LIN {X 0,Y 227.887,Z 377.096,A -85,B 0,C 180,E1 -20034.128,E2 -20034.128} C_VEL
LIN {X 0,Y 227.876,Z 377.099,A -85,B 0,C 180,E1 -20038.377,E2 -20038.377} C_VEL
LIN {X 0,Y 227.892,Z 377.098,A -85,B 0,C 180,E1 -20042.444,E2 -20042.444} C_VEL
LIN {X 0,Y 227.92,Z 377.094,A -85,B 0,C 180,E1 -20046.367,E2 -20046.367} C_VEL
LIN {X 0,Y 228.003,Z 377.201,A -85,B 0,C 180,E1 -20049.532,E2 -20049.532} C_VEL
LIN {X 0,Y 229.065,Z 380.026,A -85,B 0,C 180,E1 -20049.897,E2 -20049.897} C_VEL
LIN {X 0,Y 233.26,Z 390.63,A -85,B 0,C 180,E1 -20051.459,E2 -20051.459} C_VEL
LIN {X 0,Y 236.547,Z 400.917,A -85,B 0,C 180,E1 -20053.149,E2 -20053.149} C_VEL
LIN {X 0,Y 238.293,Z 407.679,A -85,B 0,C 180,E1 -20054.381,E2 -20054.381} C_VEL
LIN {X 0,Y 236.571,Z 418.908,A -85,B 0,C 180,E1 -20056.25,E2 -20056.25} C_VEL
LIN {X 0,Y 234.854,Z 428.795,A -85,B 0,C 180,E1 -20058.345,E2 -20058.345} C_VEL
LIN {X 0,Y 232.986,Z 438.362,A -85,B 0,C 180,E1 -20060.887,E2 -20060.887} C_VEL
LIN {X 0,Y 231.325,Z 446.044,A -85,B 0,C 180,E1 -20063.457,E2 -20063.457} C_VEL
LIN {X 0,Y 230.205,Z 451.273,A -85,B 0,C 180,E1 -20065.621,E2 -20065.621} C_VEL
LIN {X 0,Y 229.202,Z 456.365,A -85,B 0,C 180,E1 -20068.242,E2 -20068.242} C_VEL
LIN {X 0,Y 228.364,Z 460.351,A -85,B 0,C 180,E1 -20070.88,E2 -20070.88} C_VEL
LIN {X 0,Y 227.825,Z 463.315,A -85,B 0,C 180,E1 -20073.536,E2 -20073.536} C_VEL
LIN {X 0,Y 227.82,Z 464.727,A -85,B 0,C 180,E1 -20075.309,E2 -20075.309} C_VEL
LIN {X 0,Y 227.806,Z 465.754,A -85,B 0,C 180,E1 -20077.087,E2 -20077.087} C_VEL
LIN {X 0,Y 227.876,Z 466.526,A -85,B 0,C 180,E1 -20079.272,E2 -20079.272} C_VEL
LIN {X 0,Y 228.342,Z 466.545,A -85,B 0,C 180,E1 -20082.441,E2 -20082.441} C_VEL
LIN {X 0,Y 229.386,Z 465.08,A -85,B 0,C 180,E1 -20086.005,E2 -20086.005} C_VEL
LIN {X 0,Y 230.21,Z 463.745,A -85,B 0,C 180,E1 -20087.774,E2 -20087.774} C_VEL
LIN {X 0,Y 231.644,Z 460.912,A -85,B 0,C 180,E1 -20090.419,E2 -20090.419} C_VEL
LIN {X 0,Y 233.383,Z 457.03,A -85,B 0,C 180,E1 -20093.045,E2 -20093.045} C_VEL
LIN {X 0,Y 235.482,Z 451.966,A -85,B 0,C 180,E1 -20095.641,E2 -20095.641} C_VEL
LIN {X 0,Y 237.977,Z 445.525,A -85,B 0,C 180,E1 -20098.196,E2 -20098.196} C_VEL
LIN {X 0,Y 240.822,Z 437.456,A -85,B 0,C 180,E1 -20100.71,E2 -20100.71} C_VEL
LIN {X 0,Y 243.404,Z 429.151,A -85,B 0,C 180,E1 -20102.776,E2 -20102.776} C_VEL
LIN {X 0,Y 245.548,Z 421.099,A -85,B 0,C 180,E1 -20104.42,E2 -20104.42} C_VEL
LIN {X 0,Y 243.299,Z 411.924,A -85,B 0,C 180,E1 -20106.717,E2 -20106.717} C_VEL
LIN {X 0,Y 240.025,Z 402.244,A -85,B 0,C 180,E1 -20108.979,E2 -20108.979} C_VEL
LIN {X 0,Y 235.855,Z 392.708,A -85,B 0,C 180,E1 -20111.136,E2 -20111.136} C_VEL
LIN {X 0,Y 231.014,Z 383.649,A -85,B 0,C 180,E1 -20113.173,E2 -20113.173} C_VEL
LIN {X 0,Y 229.588,Z 380.946,A -85,B 0,C 180,E1 -20113.738,E2 -20113.738} C_VEL
LIN {X 0,Y 228.183,Z 378.565,A -85,B 0,C 180,E1 -20114.266,E2 -20114.266} C_VEL
LIN {X 0,Y 227.841,Z 377.102,A -85,B 0,C 180,E1 -20114.494,E2 -20114.494} C_VEL
LIN {X 0,Y 227.866,Z 377.101,A -85,B 0,C 180,E1 -20117.748,E2 -20117.748} C_VEL
LIN {X 0,Y 227.87,Z 377.105,A -85,B 0,C 180,E1 -20121.913,E2 -20121.913} C_VEL
LIN {X 0,Y 227.889,Z 377.096,A -85,B 0,C 180,E1 -20126.371,E2 -20126.371} C_VEL
LIN {X 0,Y 227.902,Z 377.05,A -85,B 0,C 180,E1 -20130.435,E2 -20130.435} C_VEL
LIN {X 0,Y 227.926,Z 377.093,A -85,B 0,C 180,E1 -20134.425,E2 -20134.425} C_VEL
LIN {X 0,Y 227.959,Z 377.082,A -85,B 0,C 180,E1 -20138.286,E2 -20138.286} C_VEL
LIN {X 0,Y 228.031,Z 377.067,A -85,B 0,C 180,E1 -20142.825,E2 -20142.825} C_VEL
LIN {X 0,Y 228.091,Z 377.072,A -85,B 0,C 180,E1 -20147.544,E2 -20147.544} C_VEL
LIN {X 0,Y 228.322,Z 377.045,A -85,B 0,C 180,E1 -20151.146,E2 -20151.146} C_VEL
LIN {X 0,Y 228.355,Z 377.031,A -85,B 0,C 180,E1 -20152.928,E2 -20152.928} C_VEL
LIN {X 0,Y 228.554,Z 377.012,A -85,B 0,C 180,E1 -20158.237,E2 -20158.237} C_VEL
LIN {X 0,Y 228.554,Z 377.013,A -85,B 0,C 180,E1 -20161.762,E2 -20161.762} C_VEL
LIN {X 0,Y 228.355,Z 377.04,A -85,B 0,C 180,E1 -20167.071,E2 -20167.071} C_VEL
LIN {X 0,Y 228.167,Z 377.054,A -85,B 0,C 180,E1 -20170.65,E2 -20170.65} C_VEL
LIN {X 0,Y 228.053,Z 377.078,A -85,B 0,C 180,E1 -20176.102,E2 -20176.102} C_VEL
LIN {X 0,Y 227.939,Z 377.091,A -85,B 0,C 180,E1 -20179.825,E2 -20179.825} C_VEL
LIN {X 0,Y 227.91,Z 377.093,A -85,B 0,C 180,E1 -20183.633,E2 -20183.633} C_VEL
LIN {X 0,Y 227.9,Z 377.101,A -85,B 0,C 180,E1 -20188.177,E2 -20188.177} C_VEL
LIN {X 0,Y 228.571,Z 380.288,A -85,B 0,C 180,E1 -20191.514,E2 -20191.514} C_VEL
LIN {X 0,Y 229.542,Z 384.592,A -85,B 0,C 180,E1 -20195.572,E2 -20195.572} C_VEL
LIN {X 0,Y 230.655,Z 390.276,A -85,B 0,C 180,E1 -20200.384,E2 -20200.384} C_VEL
LIN {X 0,Y 231.787,Z 396.318,A -85,B 0,C 180,E1 -20205.043,E2 -20205.043} C_VEL
LIN {X 0,Y 232.75,Z 401.888,A -85,B 0,C 180,E1 -20209.015,E2 -20209.015} C_VEL
LIN {X 0,Y 232.897,Z 404.605,A -85,B 0,C 180,E1 -20210.825,E2 -20210.825} C_VEL
LIN {X 0,Y 231.681,Z 409.325,A -85,B 0,C 180,E1 -20213.706,E2 -20213.706} C_VEL
LIN {X 0,Y 232.555,Z 412.987,A -85,B 0,C 180,E1 -20214.055,E2 -20214.055} C_VEL
LIN {X 0,Y 233.833,Z 417.977,A -85,B 0,C 180,E1 -20214.599,E2 -20214.599} C_VEL
LIN {X 0,Y 234.21,Z 423.584,A -85,B 0,C 180,E1 -20215.071,E2 -20215.071} C_VEL
LIN {X 0,Y 233.3,Z 433.06,A -85,B 0,C 180,E1 -20215.782,E2 -20215.782} C_VEL
LIN {X 0,Y 232.111,Z 442.304,A -85,B 0,C 180,E1 -20216.645,E2 -20216.645} C_VEL
LIN {X 0,Y 232.068,Z 447.482,A -85,B 0,C 180,E1 -20217.347,E2 -20217.347} C_VEL
LIN {X 0,Y 232.339,Z 459.542,A -85,B 0,C 180,E1 -20219.308,E2 -20219.308} C_VEL
LIN {X 0,Y 231.84,Z 470.153,A -85,B 0,C 180,E1 -20221.291,E2 -20221.291} C_VEL
LIN {X 0,Y 230.723,Z 479.469,A -85,B 0,C 180,E1 -20223.303,E2 -20223.303} C_VEL
LIN {X 0,Y 228.773,Z 488.259,A -85,B 0,C 180,E1 -20225.499,E2 -20225.499} C_VEL
LIN {X 0,Y 225.7,Z 496.785,A -85,B 0,C 180,E1 -20228.06,E2 -20228.06} C_VEL
LIN {X 0,Y 223.14,Z 504.144,A -85,B 0,C 180,E1 -20230.887,E2 -20230.887} C_VEL
LIN {X 0,Y 221.5,Z 509.326,A -85,B 0,C 180,E1 -20233.409,E2 -20233.409} C_VEL
LIN {X 0,Y 220.196,Z 513.777,A -85,B 0,C 180,E1 -20236.152,E2 -20236.152} C_VEL
LIN {X 0,Y 219.485,Z 517.195,A -85,B 0,C 180,E1 -20238.925,E2 -20238.925} C_VEL
LIN {X 0,Y 219.334,Z 520.299,A -85,B 0,C 180,E1 -20242.637,E2 -20242.637} C_VEL
LIN {X 0,Y 219.825,Z 521.726,A -85,B 0,C 180,E1 -20246.335,E2 -20246.335} C_VEL
LIN {X 0,Y 220.089,Z 521.828,A -85,B 0,C 180,E1 -20248.171,E2 -20248.171} C_VEL
LIN {X 0,Y 220.231,Z 521.508,A -85,B 0,C 180,E1 -20250.001,E2 -20250.001} C_VEL
LIN {X 0,Y 220.159,Z 520.712,A -85,B 0,C 180,E1 -20251.831,E2 -20251.831} C_VEL
LIN {X 0,Y 219.982,Z 519.453,A -85,B 0,C 180,E1 -20253.665,E2 -20253.665} C_VEL
LIN {X 0,Y 219.583,Z 515.837,A -85,B 0,C 180,E1 -20257.166,E2 -20257.166} C_VEL
LIN {X 0,Y 219.532,Z 511.426,A -85,B 0,C 180,E1 -20260.143,E2 -20260.143} C_VEL
LIN {X 0,Y 220.146,Z 505.04,A -85,B 0,C 180,E1 -20263.384,E2 -20263.384} C_VEL
LIN {X 0,Y 221.1,Z 498.086,A -85,B 0,C 180,E1 -20266.15,E2 -20266.15} C_VEL
LIN {X 0,Y 222.436,Z 491.045,A -85,B 0,C 180,E1 -20268.42,E2 -20268.42} C_VEL
LIN {X 0,Y 224.159,Z 482.585,A -85,B 0,C 180,E1 -20270.655,E2 -20270.655} C_VEL
LIN {X 0,Y 224.752,Z 475.375,A -85,B 0,C 180,E1 -20272.282,E2 -20272.282} C_VEL
LIN {X 0,Y 225.233,Z 464.959,A -85,B 0,C 180,E1 -20274.281,E2 -20274.281} C_VEL
LIN {X 0,Y 225.518,Z 453.251,A -85,B 0,C 180,E1 -20276.117,E2 -20276.117} C_VEL
LIN {X 0,Y 225.191,Z 441.055,A -85,B 0,C 180,E1 -20277.662,E2 -20277.662} C_VEL
LIN {X 0,Y 224.037,Z 427.624,A -85,B 0,C 180,E1 -20279.036,E2 -20279.036} C_VEL
LIN {X 0,Y 221.953,Z 413.948,A -85,B 0,C 180,E1 -20280.141,E2 -20280.141} C_VEL
LIN {X 0,Y 221.507,Z 411.003,A -85,B 0,C 180,E1 -20280.389,E2 -20280.389} C_VEL
LIN {X 0,Y 223.273,Z 402.178,A -85,B 0,C 180,E1 -20285.733,E2 -20285.733} C_VEL
LIN {X 0,Y 224.225,Z 397.146,A -85,B 0,C 180,E1 -20288.821,E2 -20288.821} C_VEL
LIN {X 0,Y 223.836,Z 393.482,A -85,B 0,C 180,E1 -20291.253,E2 -20291.253} C_VEL
LIN {X 0,Y 222.551,Z 386.745,A -85,B 0,C 180,E1 -20295.993,E2 -20295.993} C_VEL
LIN {X 0,Y 221.357,Z 380.661,A -85,B 0,C 180,E1 -20300.581,E2 -20300.581} C_VEL
LIN {X 0,Y 220.858,Z 377.978,A -85,B 0,C 180,E1 -20302.8,E2 -20302.8} C_VEL
LIN {X 0,Y 220.821,Z 377.981,A -85,B 0,C 180,E1 -20307.245,E2 -20307.245} C_VEL
LIN {X 0,Y 220.832,Z 377.977,A -85,B 0,C 180,E1 -20311.486,E2 -20311.486} C_VEL
LIN {X 0,Y 220.873,Z 377.974,A -85,B 0,C 180,E1 -20315.566,E2 -20315.566} C_VEL
LIN {X 0,Y 220.898,Z 377.971,A -85,B 0,C 180,E1 -20319.515,E2 -20319.515} C_VEL
LIN {X 0,Y 221.022,Z 377.955,A -85,B 0,C 180,E1 -20323.371,E2 -20323.371} C_VEL
LIN {X 0,Y 221.123,Z 377.941,A -85,B 0,C 180,E1 -20329.007,E2 -20329.007} C_VEL
LIN {X 0,Y 221.317,Z 377.917,A -85,B 0,C 180,E1 -20332.703,E2 -20332.703} C_VEL
LIN {X 0,Y 221.518,Z 377.881,A -85,B 0,C 180,E1 -20338.182,E2 -20338.182} C_VEL
LIN {X 0,Y 221.519,Z 377.89,A -85,B 0,C 180,E1 -20341.819,E2 -20341.819} C_VEL
LIN {X 0,Y 221.302,Z 377.906,A -85,B 0,C 180,E1 -20347.298,E2 -20347.298} C_VEL
LIN {X 0,Y 221.123,Z 377.939,A -85,B 0,C 180,E1 -20350.994,E2 -20350.994} C_VEL
LIN {X 0,Y 221.023,Z 377.948,A -85,B 0,C 180,E1 -20356.63,E2 -20356.63} C_VEL
LIN {X 0,Y 220.9,Z 377.965,A -85,B 0,C 180,E1 -20360.486,E2 -20360.486} C_VEL
LIN {X 0,Y 220.874,Z 377.968,A -85,B 0,C 180,E1 -20364.435,E2 -20364.435} C_VEL
LIN {X 0,Y 220.842,Z 377.972,A -85,B 0,C 180,E1 -20368.513,E2 -20368.513} C_VEL
LIN {X 0,Y 220.831,Z 377.975,A -85,B 0,C 180,E1 -20372.754,E2 -20372.754} C_VEL
LIN {X 0,Y 220.844,Z 377.976,A -85,B 0,C 180,E1 -20377.288,E2 -20377.288} C_VEL
LIN {X 0,Y 220.782,Z 377.981,A -85,B 0,C 180,E1 -20381.951,E2 -20381.951} C_VEL
LIN {X 0,Y 220.781,Z 377.983,A -85,B 0,C 180,E1 -20385.546,E2 -20385.546} C_VEL
LIN {X 0,Y 220.812,Z 377.976,A -85,B 0,C 180,E1 -20390.463,E2 -20390.463} C_VEL
LIN {X 0,Y 220.807,Z 377.979,A -85,B 0,C 180,E1 -20395.045,E2 -20395.045} C_VEL
LIN {X 0,Y 220.874,Z 377.973,A -85,B 0,C 180,E1 -20399.394,E2 -20399.394} C_VEL
LIN {X 0,Y 220.901,Z 377.969,A -85,B 0,C 180,E1 -20403.549,E2 -20403.549} C_VEL
LIN {X 0,Y 220.95,Z 378.071,A -85,B 0,C 180,E1 -20408.665,E2 -20408.665} C_VEL
LIN {X 0,Y 222.527,Z 382.229,A -85,B 0,C 180,E1 -20409.233,E2 -20409.233} C_VEL
LIN {X 0,Y 226.794,Z 393.014,A -85,B 0,C 180,E1 -20410.941,E2 -20410.941} C_VEL
LIN {X 0,Y 229.89,Z 402.635,A -85,B 0,C 180,E1 -20412.622,E2 -20412.622} C_VEL
LIN {X 0,Y 231.599,Z 409.377,A -85,B 0,C 180,E1 -20413.906,E2 -20413.906} C_VEL
LIN {X 0,Y 229.783,Z 420.479,A -85,B 0,C 180,E1 -20415.836,E2 -20415.836} C_VEL
LIN {X 0,Y 227.986,Z 430.233,A -85,B 0,C 180,E1 -20417.989,E2 -20417.989} C_VEL
LIN {X 0,Y 226.054,Z 439.706,A -85,B 0,C 180,E1 -20420.605,E2 -20420.605} C_VEL
LIN {X 0,Y 224.343,Z 447.271,A -85,B 0,C 180,E1 -20423.252,E2 -20423.252} C_VEL
LIN {X 0,Y 223.197,Z 452.453,A -85,B 0,C 180,E1 -20425.484,E2 -20425.484} C_VEL
LIN {X 0,Y 222.17,Z 457.472,A -85,B 0,C 180,E1 -20428.186,E2 -20428.186} C_VEL
LIN {X 0,Y 221.304,Z 461.404,A -85,B 0,C 180,E1 -20430.908,E2 -20430.908} C_VEL
LIN {X 0,Y 220.773,Z 464.322,A -85,B 0,C 180,E1 -20433.649,E2 -20433.649} C_VEL
LIN {X 0,Y 220.786,Z 465.69,A -85,B 0,C 180,E1 -20435.478,E2 -20435.478} C_VEL
LIN {X 0,Y 220.813,Z 467.331,A -85,B 0,C 180,E1 -20439.156,E2 -20439.156} C_VEL
LIN {X 0,Y 221.027,Z 467.571,A -85,B 0,C 180,E1 -20440.997,E2 -20440.997} C_VEL
LIN {X 0,Y 221.9,Z 466.818,A -85,B 0,C 180,E1 -20444.676,E2 -20444.676} C_VEL
LIN {X 0,Y 222.53,Z 465.869,A -85,B 0,C 180,E1 -20446.512,E2 -20446.512} C_VEL
LIN {X 0,Y 224.288,Z 462.893,A -85,B 0,C 180,E1 -20449.94,E2 -20449.94} C_VEL
LIN {X 0,Y 226.142,Z 459.077,A -85,B 0,C 180,E1 -20452.858,E2 -20452.858} C_VEL
LIN {X 0,Y 228.246,Z 454.359,A -85,B 0,C 180,E1 -20455.535,E2 -20455.535} C_VEL
LIN {X 0,Y 230.688,Z 448.476,A -85,B 0,C 180,E1 -20458.118,E2 -20458.118} C_VEL
LIN {X 0,Y 233.681,Z 440.8,A -85,B 0,C 180,E1 -20460.748,E2 -20460.748} C_VEL
LIN {X 0,Y 236.769,Z 431.449,A -85,B 0,C 180,E1 -20463.243,E2 -20463.243} C_VEL
LIN {X 0,Y 239.085,Z 423.424,A -85,B 0,C 180,E1 -20464.972,E2 -20464.972} C_VEL
LIN {X 0,Y 237.322,Z 415.381,A -85,B 0,C 180,E1 -20467.097,E2 -20467.097} C_VEL
LIN {X 0,Y 234.296,Z 405.948,A -85,B 0,C 180,E1 -20469.464,E2 -20469.464} C_VEL
LIN {X 0,Y 230.508,Z 396.85,A -85,B 0,C 180,E1 -20471.669,E2 -20471.669} C_VEL
LIN {X 0,Y 225.272,Z 386.406,A -85,B 0,C 180,E1 -20474.146,E2 -20474.146} C_VEL
LIN {X 0,Y 223.216,Z 382.634,A -85,B 0,C 180,E1 -20475.019,E2 -20475.019} C_VEL
LIN {X 0,Y 221.246,Z 379.798,A -85,B 0,C 180,E1 -20475.769,E2 -20475.769} C_VEL
LIN {X 0,Y 220.79,Z 377.984,A -85,B 0,C 180,E1 -20476.07,E2 -20476.07} C_VEL
LIN {X 0,Y 220.848,Z 377.972,A -85,B 0,C 180,E1 -20480.471,E2 -20480.471} C_VEL
LIN {X 0,Y 220.814,Z 377.979,A -85,B 0,C 180,E1 -20485.047,E2 -20485.047} C_VEL
LIN {X 0,Y 220.831,Z 377.93,A -85,B 0,C 180,E1 -20489.389,E2 -20489.389} C_VEL
LIN {X 0,Y 220.892,Z 377.965,A -85,B 0,C 180,E1 -20493.548,E2 -20493.548} C_VEL
LIN {X 0,Y 220.875,Z 377.958,A -85,B 0,C 180,E1 -20497.553,E2 -20497.553} C_VEL
LIN {X 0,Y 220.981,Z 377.944,A -85,B 0,C 180,E1 -20502.57,E2 -20502.57} C_VEL
LIN {X 0,Y 221.023,Z 377.95,A -85,B 0,C 180,E1 -20507.139,E2 -20507.139} C_VEL
LIN {X 0,Y 221.255,Z 377.925,A -85,B 0,C 180,E1 -20510.861,E2 -20510.861} C_VEL
LIN {X 0,Y 221.308,Z 377.911,A -85,B 0,C 180,E1 -20512.702,E2 -20512.702} C_VEL
LIN {X 0,Y 221.512,Z 377.889,A -85,B 0,C 180,E1 -20518.181,E2 -20518.181} C_VEL
LIN {X 0,Y 221.512,Z 377.89,A -85,B 0,C 180,E1 -20521.818,E2 -20521.818} C_VEL
LIN {X 0,Y 221.307,Z 377.919,A -85,B 0,C 180,E1 -20527.297,E2 -20527.297} C_VEL
LIN {X 0,Y 221.113,Z 377.935,A -85,B 0,C 180,E1 -20530.994,E2 -20530.994} C_VEL
LIN {X 0,Y 221.012,Z 377.951,A -85,B 0,C 180,E1 -20536.63,E2 -20536.63} C_VEL
LIN {X 0,Y 220.889,Z 377.965,A -85,B 0,C 180,E1 -20540.486,E2 -20540.486} C_VEL
LIN {X 0,Y 220.863,Z 377.973,A -85,B 0,C 180,E1 -20544.435,E2 -20544.435} C_VEL
LIN {X 0,Y 220.882,Z 378.056,A -85,B 0,C 180,E1 -20547.016,E2 -20547.016} C_VEL
LIN {X 0,Y 221.685,Z 381.884,A -85,B 0,C 180,E1 -20551.136,E2 -20551.136} C_VEL
LIN {X 0,Y 222.721,Z 386.64,A -85,B 0,C 180,E1 -20555.715,E2 -20555.715} C_VEL
LIN {X 0,Y 223.697,Z 391.587,A -85,B 0,C 180,E1 -20560.046,E2 -20560.046} C_VEL
LIN {X 0,Y 224.796,Z 397.571,A -85,B 0,C 180,E1 -20564.817,E2 -20564.817} C_VEL
LIN {X 0,Y 225.818,Z 403.494,A -85,B 0,C 180,E1 -20569.191,E2 -20569.191} C_VEL
LIN {X 0,Y 225.941,Z 405.065,A -85,B 0,C 180,E1 -20570.283,E2 -20570.283} C_VEL
LIN {X 0,Y 225.199,Z 408.146,A -85,B 0,C 180,E1 -20572.279,E2 -20572.279} C_VEL
LIN {X 0,Y 226.113,Z 412.034,A -85,B 0,C 180,E1 -20572.703,E2 -20572.703} C_VEL
LIN {X 0,Y 229.199,Z 425.135,A -85,B 0,C 180,E1 -20574.279,E2 -20574.279} C_VEL
LIN {X 0,Y 231.364,Z 438.931,A -85,B 0,C 180,E1 -20576.106,E2 -20576.106} C_VEL
LIN {X 0,Y 232.068,Z 447.482,A -85,B 0,C 180,E1 -20577.347,E2 -20577.347} C_VEL
LIN {X 0,Y 232.005,Z 451.013,A -85,B 0,C 180,E1 -20577.851,E2 -20577.851} C_VEL
LIN {X 0,Y 230.913,Z 456.25,A -85,B 0,C 180,E1 -20578.526,E2 -20578.526} C_VEL
LIN {X 0,Y 229.109,Z 461.374,A -85,B 0,C 180,E1 -20579.176,E2 -20579.176} C_VEL
LIN {X 0,Y 226.008,Z 469.424,A -85,B 0,C 180,E1 -20580.386,E2 -20580.386} C_VEL
LIN {X 0,Y 224.98,Z 473.951,A -85,B 0,C 180,E1 -20581.289,E2 -20581.289} C_VEL
LIN {X 0,Y 223.536,Z 482.712,A -85,B 0,C 180,E1 -20583.385,E2 -20583.385} C_VEL
LIN {X 0,Y 221.75,Z 489.26,A -85,B 0,C 180,E1 -20585.171,E2 -20585.171} C_VEL
LIN {X 0,Y 218.628,Z 497.453,A -85,B 0,C 180,E1 -20587.809,E2 -20587.809} C_VEL
LIN {X 0,Y 216.24,Z 503.98,A -85,B 0,C 180,E1 -20590.48,E2 -20590.48} C_VEL
LIN {X 0,Y 214.129,Z 510.227,A -85,B 0,C 180,E1 -20593.802,E2 -20593.802} C_VEL
LIN {X 0,Y 212.898,Z 514.277,A -85,B 0,C 180,E1 -20596.641,E2 -20596.641} C_VEL
LIN {X 0,Y 212.25,Z 518.145,A -85,B 0,C 180,E1 -20600.472,E2 -20600.472} C_VEL
LIN {X 0,Y 212.351,Z 519.863,A -85,B 0,C 180,E1 -20603.159,E2 -20603.159} C_VEL
LIN {X 0,Y 212.748,Z 520.857,A -85,B 0,C 180,E1 -20606.213,E2 -20606.213} C_VEL
LIN {X 0,Y 213.035,Z 520.945,A -85,B 0,C 180,E1 -20608.111,E2 -20608.111} C_VEL
LIN {X 0,Y 213.184,Z 520.605,A -85,B 0,C 180,E1 -20610.001,E2 -20610.001} C_VEL
LIN {X 0,Y 213.108,Z 519.773,A -85,B 0,C 180,E1 -20611.891,E2 -20611.891} C_VEL
LIN {X 0,Y 212.904,Z 518.49,A -85,B 0,C 180,E1 -20613.787,E2 -20613.787} C_VEL
LIN {X 0,Y 212.506,Z 515.093,A -85,B 0,C 180,E1 -20617.179,E2 -20617.179} C_VEL
LIN {X 0,Y 212.5,Z 510.36,A -85,B 0,C 180,E1 -20620.482,E2 -20620.482} C_VEL
LIN {X 0,Y 213.188,Z 503.916,A -85,B 0,C 180,E1 -20623.829,E2 -20623.829} C_VEL
LIN {X 0,Y 214.218,Z 496.905,A -85,B 0,C 180,E1 -20626.684,E2 -20626.684} C_VEL
LIN {X 0,Y 215.928,Z 488.924,A -85,B 0,C 180,E1 -20629.285,E2 -20629.285} C_VEL
LIN {X 0,Y 217.407,Z 481.258,A -85,B 0,C 180,E1 -20631.327,E2 -20631.327} C_VEL
LIN {X 0,Y 218.032,Z 471.647,A -85,B 0,C 180,E1 -20633.51,E2 -20633.51} C_VEL
LIN {X 0,Y 218.596,Z 460.828,A -85,B 0,C 180,E1 -20635.521,E2 -20635.521} C_VEL
LIN {X 0,Y 218.745,Z 449.749,A -85,B 0,C 180,E1 -20637.221,E2 -20637.221} C_VEL
LIN {X 0,Y 218.234,Z 437.493,A -85,B 0,C 180,E1 -20638.775,E2 -20638.775} C_VEL
LIN {X 0,Y 217.001,Z 424.909,A -85,B 0,C 180,E1 -20640.073,E2 -20640.073} C_VEL
LIN {X 0,Y 214.936,Z 412.402,A -85,B 0,C 180,E1 -20641.11,E2 -20641.11} C_VEL
LIN {X 0,Y 214.672,Z 410.082,A -85,B 0,C 180,E1 -20641.307,E2 -20641.307} C_VEL
LIN {X 0,Y 216.59,Z 401.221,A -85,B 0,C 180,E1 -20646.893,E2 -20646.893} C_VEL
LIN {X 0,Y 217.178,Z 397.839,A -85,B 0,C 180,E1 -20649.045,E2 -20649.045} C_VEL
LIN {X 0,Y 216.714,Z 393.929,A -85,B 0,C 180,E1 -20651.765,E2 -20651.765} C_VEL
LIN {X 0,Y 215.394,Z 387.122,A -85,B 0,C 180,E1 -20656.749,E2 -20656.749} C_VEL
LIN {X 0,Y 214.269,Z 381.185,A -85,B 0,C 180,E1 -20661.45,E2 -20661.45} C_VEL
LIN {X 0,Y 213.765,Z 378.863,A -85,B 0,C 180,E1 -20663.49,E2 -20663.49} C_VEL
LIN {X 0,Y 213.772,Z 378.857,A -85,B 0,C 180,E1 -20668.263,E2 -20668.263} C_VEL
LIN {X 0,Y 213.831,Z 378.852,A -85,B 0,C 180,E1 -20672.604,E2 -20672.604} C_VEL
LIN {X 0,Y 213.857,Z 378.851,A -85,B 0,C 180,E1 -20676.954,E2 -20676.954} C_VEL
LIN {X 0,Y 213.938,Z 378.84,A -85,B 0,C 180,E1 -20682.306,E2 -20682.306} C_VEL
LIN {X 0,Y 213.987,Z 378.831,A -85,B 0,C 180,E1 -20686.709,E2 -20686.709} C_VEL
LIN {X 0,Y 214.203,Z 378.805,A -85,B 0,C 180,E1 -20690.558,E2 -20690.558} C_VEL
LIN {X 0,Y 214.254,Z 378.797,A -85,B 0,C 180,E1 -20692.461,E2 -20692.461} C_VEL
LIN {X 0,Y 214.452,Z 378.761,A -85,B 0,C 180,E1 -20698.122,E2 -20698.122} C_VEL
LIN {X 0,Y 214.557,Z 378.751,A -85,B 0,C 180,E1 -20700,E2 -20700} C_VEL
LIN {X 0,Y 214.452,Z 378.77,A -85,B 0,C 180,E1 -20701.878,E2 -20701.878} C_VEL
LIN {X 0,Y 214.242,Z 378.785,A -85,B 0,C 180,E1 -20707.54,E2 -20707.54} C_VEL
LIN {X 0,Y 214.054,Z 378.82,A -85,B 0,C 180,E1 -20711.362,E2 -20711.362} C_VEL
LIN {X 0,Y 213.94,Z 378.823,A -85,B 0,C 180,E1 -20715.237,E2 -20715.237} C_VEL
LIN {X 0,Y 213.847,Z 378.846,A -85,B 0,C 180,E1 -20719.187,E2 -20719.187} C_VEL
LIN {X 0,Y 213.854,Z 378.835,A -85,B 0,C 180,E1 -20723.227,E2 -20723.227} C_VEL
LIN {X 0,Y 213.835,Z 378.85,A -85,B 0,C 180,E1 -20727.45,E2 -20727.45} C_VEL
LIN {X 0,Y 213.786,Z 378.851,A -85,B 0,C 180,E1 -20731.735,E2 -20731.735} C_VEL
LIN {X 0,Y 213.759,Z 378.857,A -85,B 0,C 180,E1 -20736.286,E2 -20736.286} C_VEL
LIN {X 0,Y 213.724,Z 378.862,A -85,B 0,C 180,E1 -20741.123,E2 -20741.123} C_VEL
LIN {X 0,Y 213.715,Z 378.861,A -85,B 0,C 180,E1 -20743.677,E2 -20743.677} C_VEL
LIN {X 0,Y 213.713,Z 378.861,A -85,B 0,C 180,E1 -20746.343,E2 -20746.343} C_VEL
LIN {X 0,Y 213.723,Z 378.862,A -85,B 0,C 180,E1 -20749.142,E2 -20749.142} C_VEL
LIN {X 0,Y 213.749,Z 378.858,A -85,B 0,C 180,E1 -20753.711,E2 -20753.711} C_VEL
LIN {X 0,Y 213.801,Z 378.853,A -85,B 0,C 180,E1 -20758.724,E2 -20758.724} C_VEL
LIN {X 0,Y 213.832,Z 378.85,A -85,B 0,C 180,E1 -20762.602,E2 -20762.602} C_VEL
LIN {X 0,Y 213.874,Z 378.981,A -85,B 0,C 180,E1 -20767.734,E2 -20767.734} C_VEL
LIN {X 0,Y 215.527,Z 383.212,A -85,B 0,C 180,E1 -20768.351,E2 -20768.351} C_VEL
LIN {X 0,Y 219.732,Z 393.58,A -85,B 0,C 180,E1 -20770.08,E2 -20770.08} C_VEL
LIN {X 0,Y 223.224,Z 404.275,A -85,B 0,C 180,E1 -20772.047,E2 -20772.047} C_VEL
LIN {X 0,Y 224.901,Z 411.091,A -85,B 0,C 180,E1 -20773.402,E2 -20773.402} C_VEL
LIN {X 0,Y 223.205,Z 420.972,A -85,B 0,C 180,E1 -20775.176,E2 -20775.176} C_VEL
LIN {X 0,Y 221.5,Z 429.918,A -85,B 0,C 180,E1 -20777.166,E2 -20777.166} C_VEL
LIN {X 0,Y 219.435,Z 439.59,A -85,B 0,C 180,E1 -20779.853,E2 -20779.853} C_VEL
LIN {X 0,Y 217.609,Z 447.39,A -85,B 0,C 180,E1 -20782.576,E2 -20782.576} C_VEL
LIN {X 0,Y 216.19,Z 453.613,A -85,B 0,C 180,E1 -20785.337,E2 -20785.337} C_VEL
LIN {X 0,Y 215.138,Z 458.568,A -85,B 0,C 180,E1 -20788.127,E2 -20788.127} C_VEL
LIN {X 0,Y 214.214,Z 462.452,A -85,B 0,C 180,E1 -20790.939,E2 -20790.939} C_VEL
LIN {X 0,Y 213.721,Z 465.314,A -85,B 0,C 180,E1 -20793.77,E2 -20793.77} C_VEL
LIN {X 0,Y 213.733,Z 466.656,A -85,B 0,C 180,E1 -20795.66,E2 -20795.66} C_VEL
LIN {X 0,Y 213.818,Z 468.245,A -85,B 0,C 180,E1 -20799.458,E2 -20799.458} C_VEL
LIN {X 0,Y 214.05,Z 468.437,A -85,B 0,C 180,E1 -20801.36,E2 -20801.36} C_VEL
LIN {X 0,Y 214.99,Z 467.635,A -85,B 0,C 180,E1 -20805.159,E2 -20805.159} C_VEL
LIN {X 0,Y 215.693,Z 466.658,A -85,B 0,C 180,E1 -20807.051,E2 -20807.051} C_VEL
LIN {X 0,Y 217.449,Z 463.811,A -85,B 0,C 180,E1 -20810.397,E2 -20810.397} C_VEL
LIN {X 0,Y 219.556,Z 459.729,A -85,B 0,C 180,E1 -20813.585,E2 -20813.585} C_VEL
LIN {X 0,Y 221.795,Z 454.948,A -85,B 0,C 180,E1 -20816.333,E2 -20816.333} C_VEL
LIN {X 0,Y 224.464,Z 448.867,A -85,B 0,C 180,E1 -20819.03,E2 -20819.03} C_VEL
LIN {X 0,Y 227.536,Z 441.205,A -85,B 0,C 180,E1 -20821.673,E2 -20821.673} C_VEL
LIN {X 0,Y 230.722,Z 432,A -85,B 0,C 180,E1 -20824.159,E2 -20824.159} C_VEL
LIN {X 0,Y 232.598,Z 425.841,A -85,B 0,C 180,E1 -20825.54,E2 -20825.54} C_VEL
LIN {X 0,Y 232.422,Z 423.825,A -85,B 0,C 180,E1 -20826.081,E2 -20826.081} C_VEL
LIN {X 0,Y 230.339,Z 415.343,A -85,B 0,C 180,E1 -20828.443,E2 -20828.443} C_VEL
LIN {X 0,Y 227.414,Z 406.442,A -85,B 0,C 180,E1 -20830.784,E2 -20830.784} C_VEL
LIN {X 0,Y 223.373,Z 397.204,A -85,B 0,C 180,E1 -20833.184,E2 -20833.184} C_VEL
LIN {X 0,Y 219.378,Z 389.416,A -85,B 0,C 180,E1 -20835.186,E2 -20835.186} C_VEL
LIN {X 0,Y 218.363,Z 387.299,A -85,B 0,C 180,E1 -20835.694,E2 -20835.694} C_VEL
LIN {X 0,Y 216.407,Z 384.047,A -85,B 0,C 180,E1 -20836.548,E2 -20836.548} C_VEL
LIN {X 0,Y 215.374,Z 382.529,A -85,B 0,C 180,E1 -20836.978,E2 -20836.978} C_VEL
LIN {X 0,Y 213.981,Z 379.934,A -85,B 0,C 180,E1 -20837.597,E2 -20837.597} C_VEL
LIN {X 0,Y 213.786,Z 378.855,A -85,B 0,C 180,E1 -20837.788,E2 -20837.788} C_VEL
LIN {X 0,Y 213.779,Z 378.859,A -85,B 0,C 180,E1 -20842.09,E2 -20842.09} C_VEL
LIN {X 0,Y 213.768,Z 378.857,A -85,B 0,C 180,E1 -20846.019,E2 -20846.019} C_VEL
LIN {X 0,Y 213.758,Z 378.81,A -85,B 0,C 180,E1 -20850.45,E2 -20850.45} C_VEL
LIN {X 0,Y 213.799,Z 378.852,A -85,B 0,C 180,E1 -20854.701,E2 -20854.701} C_VEL
LIN {X 0,Y 213.81,Z 378.849,A -85,B 0,C 180,E1 -20858.803,E2 -20858.803} C_VEL
LIN {X 0,Y 213.941,Z 378.821,A -85,B 0,C 180,E1 -20862.803,E2 -20862.803} C_VEL
LIN {X 0,Y 213.978,Z 378.827,A -85,B 0,C 180,E1 -20866.708,E2 -20866.708} C_VEL
LIN {X 0,Y 214.193,Z 378.802,A -85,B 0,C 180,E1 -20870.557,E2 -20870.557} C_VEL
LIN {X 0,Y 214.245,Z 378.793,A -85,B 0,C 180,E1 -20872.46,E2 -20872.46} C_VEL
LIN {X 0,Y 214.446,Z 378.77,A -85,B 0,C 180,E1 -20878.121,E2 -20878.121} C_VEL
LIN {X 0,Y 214.552,Z 378.744,A -85,B 0,C 180,E1 -20880,E2 -20880} C_VEL
LIN {X 0,Y 214.445,Z 378.771,A -85,B 0,C 180,E1 -20881.878,E2 -20881.878} C_VEL
LIN {X 0,Y 214.244,Z 378.799,A -85,B 0,C 180,E1 -20887.539,E2 -20887.539} C_VEL
LIN {X 0,Y 214.043,Z 378.82,A -85,B 0,C 180,E1 -20891.362,E2 -20891.362} C_VEL
LIN {X 0,Y 213.93,Z 378.833,A -85,B 0,C 180,E1 -20895.237,E2 -20895.237} C_VEL
LIN {X 0,Y 213.864,Z 378.847,A -85,B 0,C 180,E1 -20899.185,E2 -20899.185} C_VEL
LIN {X 0,Y 213.843,Z 378.846,A -85,B 0,C 180,E1 -20903.227,E2 -20903.227} C_VEL
LIN {X 0,Y 213.807,Z 378.9,A -85,B 0,C 180,E1 -20905.558,E2 -20905.558} C_VEL
LIN {X 0,Y 214.767,Z 383.21,A -85,B 0,C 180,E1 -20910.478,E2 -20910.478} C_VEL
LIN {X 0,Y 215.812,Z 388.242,A -85,B 0,C 180,E1 -20915.5,E2 -20915.5} C_VEL
LIN {X 0,Y 216.874,Z 393.695,A -85,B 0,C 180,E1 -20920.4,E2 -20920.4} C_VEL
LIN {X 0,Y 217.957,Z 399.561,A -85,B 0,C 180,E1 -20925.185,E2 -20925.185} C_VEL
LIN {X 0,Y 218.791,Z 404.452,A -85,B 0,C 180,E1 -20928.91,E2 -20928.91} C_VEL
LIN {X 0,Y 218.763,Z 407.134,A -85,B 0,C 180,E1 -20930.806,E2 -20930.806} C_VEL
LIN {X 0,Y 219.811,Z 411.225,A -85,B 0,C 180,E1 -20931.284,E2 -20931.284} C_VEL
LIN {X 0,Y 222.805,Z 423.827,A -85,B 0,C 180,E1 -20932.896,E2 -20932.896} C_VEL
LIN {X 0,Y 224.805,Z 436.288,A -85,B 0,C 180,E1 -20934.619,E2 -20934.619} C_VEL
LIN {X 0,Y 225.713,Z 446.531,A -85,B 0,C 180,E1 -20936.165,E2 -20936.165} C_VEL
LIN {X 0,Y 226.018,Z 457.903,A -85,B 0,C 180,E1 -20938.09,E2 -20938.09} C_VEL
LIN {X 0,Y 225.428,Z 469.4,A -85,B 0,C 180,E1 -20940.304,E2 -20940.304} C_VEL
LIN {X 0,Y 224.98,Z 473.951,A -85,B 0,C 180,E1 -20941.289,E2 -20941.289} C_VEL
LIN {X 0,Y 223.761,Z 478.385,A -85,B 0,C 180,E1 -20942.234,E2 -20942.234} C_VEL
LIN {X 0,Y 221.418,Z 482.633,A -85,B 0,C 180,E1 -20943.124,E2 -20943.124} C_VEL
LIN {X 0,Y 214.721,Z 491.717,A -85,B 0,C 180,E1 -20945.339,E2 -20945.339} C_VEL
LIN {X 0,Y 212.666,Z 495.3,A -85,B 0,C 180,E1 -20946.511,E2 -20946.511} C_VEL
LIN {X 0,Y 209.87,Z 502.432,A -85,B 0,C 180,E1 -20949.416,E2 -20949.416} C_VEL
LIN {X 0,Y 207.84,Z 507.943,A -85,B 0,C 180,E1 -20952.284,E2 -20952.284} C_VEL
LIN {X 0,Y 206.326,Z 512.301,A -85,B 0,C 180,E1 -20955.2,E2 -20955.2} C_VEL
LIN {X 0,Y 205.438,Z 515.633,A -85,B 0,C 180,E1 -20958.157,E2 -20958.157} C_VEL
LIN {X 0,Y 205.202,Z 517.347,A -85,B 0,C 180,E1 -20960.141,E2 -20960.141} C_VEL
LIN {X 0,Y 205.297,Z 519.115,A -85,B 0,C 180,E1 -20963.103,E2 -20963.103} C_VEL
LIN {X 0,Y 205.673,Z 519.988,A -85,B 0,C 180,E1 -20966.083,E2 -20966.083} C_VEL
LIN {X 0,Y 205.98,Z 520.062,A -85,B 0,C 180,E1 -20968.046,E2 -20968.046} C_VEL
LIN {X 0,Y 206.137,Z 519.694,A -85,B 0,C 180,E1 -20970.001,E2 -20970.001} C_VEL
LIN {X 0,Y 206.056,Z 518.833,A -85,B 0,C 180,E1 -20971.956,E2 -20971.956} C_VEL
LIN {X 0,Y 205.827,Z 517.526,A -85,B 0,C 180,E1 -20973.917,E2 -20973.917} C_VEL
LIN {X 0,Y 205.428,Z 514.347,A -85,B 0,C 180,E1 -20977.191,E2 -20977.191} C_VEL
LIN {X 0,Y 205.458,Z 509.278,A -85,B 0,C 180,E1 -20980.845,E2 -20980.845} C_VEL
LIN {X 0,Y 206.234,Z 502.785,A -85,B 0,C 180,E1 -20984.305,E2 -20984.305} C_VEL
LIN {X 0,Y 207.358,Z 495.719,A -85,B 0,C 180,E1 -20987.253,E2 -20987.253} C_VEL
LIN {X 0,Y 209.278,Z 487.132,A -85,B 0,C 180,E1 -20990.084,E2 -20990.084} C_VEL
LIN {X 0,Y 210.607,Z 479.902,A -85,B 0,C 180,E1 -20992.051,E2 -20992.051} C_VEL
LIN {X 0,Y 211.29,Z 468.9,A -85,B 0,C 180,E1 -20994.57,E2 -20994.57} C_VEL
LIN {X 0,Y 211.892,Z 457.844,A -85,B 0,C 180,E1 -20996.625,E2 -20996.625} C_VEL
LIN {X 0,Y 211.962,Z 446.75,A -85,B 0,C 180,E1 -20998.331,E2 -20998.331} C_VEL
LIN {X 0,Y 211.336,Z 434.126,A -85,B 0,C 180,E1 -20999.924,E2 -20999.924} C_VEL
LIN {X 0,Y 209.856,Z 421.01,A -85,B 0,C 180,E1 -21001.266,E2 -21001.266} C_VEL
LIN {X 0,Y 207.846,Z 409.211,A -85,B 0,C 180,E1 -21002.292,E2 -21002.292} C_VEL
LIN {X 0,Y 209.579,Z 401.801,A -85,B 0,C 180,E1 -21007.131,E2 -21007.131} C_VEL
LIN {X 0,Y 210.103,Z 398.313,A -85,B 0,C 180,E1 -21009.463,E2 -21009.463} C_VEL
LIN {X 0,Y 209.533,Z 394.15,A -85,B 0,C 180,E1 -21012.447,E2 -21012.447} C_VEL
LIN {X 0,Y 208.555,Z 389.095,A -85,B 0,C 180,E1 -21016.305,E2 -21016.305} C_VEL
LIN {X 0,Y 207.39,Z 383.072,A -85,B 0,C 180,E1 -21021.21,E2 -21021.21} C_VEL
LIN {X 0,Y 206.708,Z 379.741,A -85,B 0,C 180,E1 -21024.258,E2 -21024.258} C_VEL
LIN {X 0,Y 206.711,Z 379.737,A -85,B 0,C 180,E1 -21029.337,E2 -21029.337} C_VEL
LIN {X 0,Y 206.738,Z 379.734,A -85,B 0,C 180,E1 -21033.773,E2 -21033.773} C_VEL
LIN {X 0,Y 206.763,Z 379.733,A -85,B 0,C 180,E1 -21038.044,E2 -21038.044} C_VEL
LIN {X 0,Y 206.882,Z 379.719,A -85,B 0,C 180,E1 -21042.198,E2 -21042.198} C_VEL
LIN {X 0,Y 206.92,Z 379.713,A -85,B 0,C 180,E1 -21046.246,E2 -21046.246} C_VEL
LIN {X 0,Y 207.139,Z 379.684,A -85,B 0,C 180,E1 -21050.233,E2 -21050.233} C_VEL
LIN {X 0,Y 207.195,Z 379.677,A -85,B 0,C 180,E1 -21052.203,E2 -21052.203} C_VEL
LIN {X 0,Y 207.388,Z 379.64,A -85,B 0,C 180,E1 -21058.058,E2 -21058.058} C_VEL
LIN {X 0,Y 207.522,Z 379.627,A -85,B 0,C 180,E1 -21060,E2 -21060} C_VEL
LIN {X 0,Y 207.389,Z 379.651,A -85,B 0,C 180,E1 -21061.942,E2 -21061.942} C_VEL
LIN {X 0,Y 207.185,Z 379.665,A -85,B 0,C 180,E1 -21067.799,E2 -21067.799} C_VEL
LIN {X 0,Y 206.99,Z 379.702,A -85,B 0,C 180,E1 -21071.755,E2 -21071.755} C_VEL
LIN {X 0,Y 206.873,Z 379.704,A -85,B 0,C 180,E1 -21075.771,E2 -21075.771} C_VEL
LIN {X 0,Y 206.791,Z 379.726,A -85,B 0,C 180,E1 -21079.869,E2 -21079.869} C_VEL
LIN {X 0,Y 206.77,Z 379.722,A -85,B 0,C 180,E1 -21084.072,E2 -21084.072} C_VEL
LIN {X 0,Y 206.75,Z 379.727,A -85,B 0,C 180,E1 -21088.418,E2 -21088.418} C_VEL
LIN {X 0,Y 206.716,Z 379.734,A -85,B 0,C 180,E1 -21092.955,E2 -21092.955} C_VEL
LIN {X 0,Y 206.728,Z 379.733,A -85,B 0,C 180,E1 -21095.32,E2 -21095.32} C_VEL
LIN {X 0,Y 206.673,Z 379.739,A -85,B 0,C 180,E1 -21100.249,E2 -21100.249} C_VEL
LIN {X 0,Y 206.642,Z 379.74,A -85,B 0,C 180,E1 -21104.419,E2 -21104.419} C_VEL
LIN {X 0,Y 206.648,Z 379.741,A -85,B 0,C 180,E1 -21108.436,E2 -21108.436} C_VEL
LIN {X 0,Y 206.686,Z 379.735,A -85,B 0,C 180,E1 -21112.26,E2 -21112.26} C_VEL
LIN {X 0,Y 206.708,Z 379.736,A -85,B 0,C 180,E1 -21117.042,E2 -21117.042} C_VEL
LIN {X 0,Y 206.772,Z 379.729,A -85,B 0,C 180,E1 -21122.096,E2 -21122.096} C_VEL
LIN {X 0,Y 206.854,Z 379.893,A -85,B 0,C 180,E1 -21126.74,E2 -21126.74} C_VEL
LIN {X 0,Y 207.905,Z 382.675,A -85,B 0,C 180,E1 -21127.161,E2 -21127.161} C_VEL
LIN {X 0,Y 212.651,Z 394.071,A -85,B 0,C 180,E1 -21129.144,E2 -21129.144} C_VEL
LIN {X 0,Y 215.966,Z 403.815,A -85,B 0,C 180,E1 -21131.007,E2 -21131.007} C_VEL
LIN {X 0,Y 218.221,Z 412.792,A -85,B 0,C 180,E1 -21132.87,E2 -21132.87} C_VEL
LIN {X 0,Y 216.236,Z 423.578,A -85,B 0,C 180,E1 -21134.928,E2 -21134.928} C_VEL
LIN {X 0,Y 214.327,Z 433.099,A -85,B 0,C 180,E1 -21137.211,E2 -21137.211} C_VEL
LIN {X 0,Y 212.524,Z 440.934,A -85,B 0,C 180,E1 -21139.519,E2 -21139.519} C_VEL
LIN {X 0,Y 210.641,Z 448.626,A -85,B 0,C 180,E1 -21142.329,E2 -21142.329} C_VEL
LIN {X 0,Y 209.184,Z 454.771,A -85,B 0,C 180,E1 -21145.18,E2 -21145.18} C_VEL
LIN {X 0,Y 208.082,Z 459.669,A -85,B 0,C 180,E1 -21148.063,E2 -21148.063} C_VEL
LIN {X 0,Y 207.132,Z 463.498,A -85,B 0,C 180,E1 -21150.971,E2 -21150.971} C_VEL
LIN {X 0,Y 206.667,Z 466.303,A -85,B 0,C 180,E1 -21153.898,E2 -21153.898} C_VEL
LIN {X 0,Y 206.683,Z 467.621,A -85,B 0,C 180,E1 -21155.854,E2 -21155.854} C_VEL
LIN {X 0,Y 206.821,Z 469.152,A -85,B 0,C 180,E1 -21159.781,E2 -21159.781} C_VEL
LIN {X 0,Y 207.528,Z 469.065,A -85,B 0,C 180,E1 -21163.711,E2 -21163.711} C_VEL
LIN {X 0,Y 208.102,Z 468.452,A -85,B 0,C 180,E1 -21165.673,E2 -21165.673} C_VEL
LIN {X 0,Y 208.874,Z 467.436,A -85,B 0,C 180,E1 -21167.626,E2 -21167.626} C_VEL
LIN {X 0,Y 210.668,Z 464.689,A -85,B 0,C 180,E1 -21170.916,E2 -21170.916} C_VEL
LIN {X 0,Y 213.011,Z 460.381,A -85,B 0,C 180,E1 -21174.355,E2 -21174.355} C_VEL
LIN {X 0,Y 215.392,Z 455.539,A -85,B 0,C 180,E1 -21177.18,E2 -21177.18} C_VEL
LIN {X 0,Y 218.135,Z 449.607,A -85,B 0,C 180,E1 -21179.851,E2 -21179.851} C_VEL
LIN {X 0,Y 220.91,Z 443.041,A -85,B 0,C 180,E1 -21182.199,E2 -21182.199} C_VEL
LIN {X 0,Y 223.782,Z 435.375,A -85,B 0,C 180,E1 -21184.422,E2 -21184.422} C_VEL
LIN {X 0,Y 226.206,Z 427.995,A -85,B 0,C 180,E1 -21186.177,E2 -21186.177} C_VEL
LIN {X 0,Y 225.685,Z 424.084,A -85,B 0,C 180,E1 -21187.329,E2 -21187.329} C_VEL
LIN {X 0,Y 223.415,Z 415.144,A -85,B 0,C 180,E1 -21189.926,E2 -21189.926} C_VEL
LIN {X 0,Y 220.555,Z 407.022,A -85,B 0,C 180,E1 -21192.194,E2 -21192.194} C_VEL
LIN {X 0,Y 216.062,Z 397.042,A -85,B 0,C 180,E1 -21194.969,E2 -21194.969} C_VEL
LIN {X 0,Y 211.882,Z 389.086,A -85,B 0,C 180,E1 -21197.156,E2 -21197.156} C_VEL
LIN {X 0,Y 209.472,Z 384.859,A -85,B 0,C 180,E1 -21198.325,E2 -21198.325} C_VEL
LIN {X 0,Y 207.173,Z 381.5,A -85,B 0,C 180,E1 -21199.35,E2 -21199.35} C_VEL
LIN {X 0,Y 206.704,Z 379.734,A -85,B 0,C 180,E1 -21199.684,E2 -21199.684} C_VEL
LIN {X 0,Y 206.722,Z 379.737,A -85,B 0,C 180,E1 -21202.268,E2 -21202.268} C_VEL
LIN {X 0,Y 206.704,Z 379.719,A -85,B 0,C 180,E1 -21207.043,E2 -21207.043} C_VEL
LIN {X 0,Y 206.762,Z 379.698,A -85,B 0,C 180,E1 -21212.096,E2 -21212.096} C_VEL
LIN {X 0,Y 206.783,Z 379.712,A -85,B 0,C 180,E1 -21216.583,E2 -21216.583} C_VEL
LIN {X 0,Y 206.87,Z 379.7,A -85,B 0,C 180,E1 -21222.196,E2 -21222.196} C_VEL
LIN {X 0,Y 206.911,Z 379.708,A -85,B 0,C 180,E1 -21226.245,E2 -21226.245} C_VEL
LIN {X 0,Y 207.129,Z 379.68,A -85,B 0,C 180,E1 -21230.232,E2 -21230.232} C_VEL
LIN {X 0,Y 207.185,Z 379.674,A -85,B 0,C 180,E1 -21232.201,E2 -21232.201} C_VEL
LIN {X 0,Y 207.382,Z 379.65,A -85,B 0,C 180,E1 -21238.057,E2 -21238.057} C_VEL
LIN {X 0,Y 207.516,Z 379.62,A -85,B 0,C 180,E1 -21240,E2 -21240} C_VEL
LIN {X 0,Y 207.086,Z 379.682,A -85,B 0,C 180,E1 -21243.892,E2 -21243.892} C_VEL
LIN {X 0,Y 207.185,Z 379.678,A -85,B 0,C 180,E1 -21247.798,E2 -21247.798} C_VEL
LIN {X 0,Y 206.979,Z 379.702,A -85,B 0,C 180,E1 -21251.755,E2 -21251.755} C_VEL
LIN {X 0,Y 206.864,Z 379.718,A -85,B 0,C 180,E1 -21255.771,E2 -21255.771} C_VEL
LIN {X 0,Y 206.796,Z 379.724,A -85,B 0,C 180,E1 -21259.868,E2 -21259.868} C_VEL
LIN {X 0,Y 206.758,Z 379.819,A -85,B 0,C 180,E1 -21264.072,E2 -21264.072} C_VEL
LIN {X 0,Y 207.498,Z 383.245,A -85,B 0,C 180,E1 -21268.306,E2 -21268.306} C_VEL
LIN {X 0,Y 207.953,Z 385.17,A -85,B 0,C 180,E1 -21270.46,E2 -21270.46} C_VEL
LIN {X 0,Y 208.823,Z 389.482,A -85,B 0,C 180,E1 -21274.899,E2 -21274.899} C_VEL
LIN {X 0,Y 209.786,Z 394.5,A -85,B 0,C 180,E1 -21279.602,E2 -21279.602} C_VEL
LIN {X 0,Y 210.868,Z 400.128,A -85,B 0,C 180,E1 -21284.419,E2 -21284.419} C_VEL
LIN {X 0,Y 211.86,Z 406.101,A -85,B 0,C 180,E1 -21289.074,E2 -21289.074} C_VEL
LIN {X 0,Y 213.073,Z 409.648,A -85,B 0,C 180,E1 -21289.581,E2 -21289.581} C_VEL
LIN {X 0,Y 213.954,Z 411.941,A -85,B 0,C 180,E1 -21289.958,E2 -21289.958} C_VEL
LIN {X 0,Y 216.966,Z 424.962,A -85,B 0,C 180,E1 -21291.768,E2 -21291.768} C_VEL
LIN {X 0,Y 218.799,Z 437.459,A -85,B 0,C 180,E1 -21293.613,E2 -21293.613} C_VEL
LIN {X 0,Y 219.572,Z 448.197,A -85,B 0,C 180,E1 -21295.348,E2 -21295.348} C_VEL
LIN {X 0,Y 219.662,Z 459.157,A -85,B 0,C 180,E1 -21297.324,E2 -21297.324} C_VEL
LIN {X 0,Y 218.933,Z 469.94,A -85,B 0,C 180,E1 -21299.534,E2 -21299.534} C_VEL
LIN {X 0,Y 217.756,Z 478.602,A -85,B 0,C 180,E1 -21301.574,E2 -21301.574} C_VEL
LIN {X 0,Y 216.221,Z 485.609,A -85,B 0,C 180,E1 -21303.455,E2 -21303.455} C_VEL
LIN {X 0,Y 213.596,Z 493.011,A -85,B 0,C 180,E1 -21305.716,E2 -21305.716} C_VEL
LIN {X 0,Y 212.666,Z 495.3,A -85,B 0,C 180,E1 -21306.511,E2 -21306.511} C_VEL
LIN {X 0,Y 210.664,Z 498.646,A -85,B 0,C 180,E1 -21307.729,E2 -21307.729} C_VEL
LIN {X 0,Y 205.926,Z 503.494,A -85,B 0,C 180,E1 -21309.731,E2 -21309.731} C_VEL
LIN {X 0,Y 201.503,Z 507.661,A -85,B 0,C 180,E1 -21311.927,E2 -21311.927} C_VEL
LIN {X 0,Y 200.025,Z 509.89,A -85,B 0,C 180,E1 -21313.415,E2 -21313.415} C_VEL
LIN {X 0,Y 198.678,Z 513.881,A -85,B 0,C 180,E1 -21316.709,E2 -21316.709} C_VEL
LIN {X 0,Y 198.148,Z 516.546,A -85,B 0,C 180,E1 -21319.787,E2 -21319.787} C_VEL
LIN {X 0,Y 198.288,Z 518.655,A -85,B 0,C 180,E1 -21323.898,E2 -21323.898} C_VEL
LIN {X 0,Y 198.601,Z 519.12,A -85,B 0,C 180,E1 -21325.943,E2 -21325.943} C_VEL
LIN {X 0,Y 198.924,Z 519.178,A -85,B 0,C 180,E1 -21327.977,E2 -21327.977} C_VEL
LIN {X 0,Y 199.091,Z 518.775,A -85,B 0,C 180,E1 -21330.001,E2 -21330.001} C_VEL
LIN {X 0,Y 199.002,Z 517.892,A -85,B 0,C 180,E1 -21332.025,E2 -21332.025} C_VEL
LIN {X 0,Y 198.751,Z 516.561,A -85,B 0,C 180,E1 -21334.057,E2 -21334.057} C_VEL
LIN {X 0,Y 198.368,Z 513.558,A -85,B 0,C 180,E1 -21337.246,E2 -21337.246} C_VEL
LIN {X 0,Y 198.329,Z 509.75,A -85,B 0,C 180,E1 -21340.207,E2 -21340.207} C_VEL
LIN {X 0,Y 198.841,Z 504.669,A -85,B 0,C 180,E1 -21343.283,E2 -21343.283} C_VEL
LIN {X 0,Y 199.799,Z 498.277,A -85,B 0,C 180,E1 -21346.345,E2 -21346.345} C_VEL
LIN {X 0,Y 201.166,Z 491.529,A -85,B 0,C 180,E1 -21348.949,E2 -21348.949} C_VEL
LIN {X 0,Y 202.99,Z 484.021,A -85,B 0,C 180,E1 -21351.319,E2 -21351.319} C_VEL
LIN {X 0,Y 203.911,Z 476.454,A -85,B 0,C 180,E1 -21353.352,E2 -21353.352} C_VEL
LIN {X 0,Y 204.656,Z 466.16,A -85,B 0,C 180,E1 -21355.695,E2 -21355.695} C_VEL
LIN {X 0,Y 205.194,Z 455.775,A -85,B 0,C 180,E1 -21357.639,E2 -21357.639} C_VEL
LIN {X 0,Y 205.204,Z 444.086,A -85,B 0,C 180,E1 -21359.45,E2 -21359.45} C_VEL
LIN {X 0,Y 204.514,Z 431.71,A -85,B 0,C 180,E1 -21361.03,E2 -21361.03} C_VEL
LIN {X 0,Y 202.907,Z 418.86,A -85,B 0,C 180,E1 -21362.393,E2 -21362.393} C_VEL
LIN {X 0,Y 201.074,Z 408.294,A -85,B 0,C 180,E1 -21363.36,E2 -21363.36} C_VEL
LIN {X 0,Y 202.674,Z 401.91,A -85,B 0,C 180,E1 -21367.695,E2 -21367.695} C_VEL
LIN {X 0,Y 203.048,Z 399.395,A -85,B 0,C 180,E1 -21369.446,E2 -21369.446} C_VEL
LIN {X 0,Y 202.585,Z 395.672,A -85,B 0,C 180,E1 -21372.183,E2 -21372.183} C_VEL
LIN {X 0,Y 201.706,Z 391.043,A -85,B 0,C 180,E1 -21375.825,E2 -21375.825} C_VEL
LIN {X 0,Y 200.622,Z 385.542,A -85,B 0,C 180,E1 -21380.418,E2 -21380.418} C_VEL
LIN {X 0,Y 199.693,Z 380.616,A -85,B 0,C 180,E1 -21384.851,E2 -21384.851} C_VEL
LIN {X 0,Y 199.698,Z 380.61,A -85,B 0,C 180,E1 -21388.137,E2 -21388.137} C_VEL
LIN {X 0,Y 199.691,Z 380.613,A -85,B 0,C 180,E1 -21392.773,E2 -21392.773} C_VEL
LIN {X 0,Y 199.743,Z 380.608,A -85,B 0,C 180,E1 -21397.23,E2 -21397.23} C_VEL
LIN {X 0,Y 199.843,Z 380.595,A -85,B 0,C 180,E1 -21401.723,E2 -21401.723} C_VEL
LIN {X 0,Y 199.854,Z 380.592,A -85,B 0,C 180,E1 -21405.75,E2 -21405.75} C_VEL
LIN {X 0,Y 200.082,Z 380.562,A -85,B 0,C 180,E1 -21409.885,E2 -21409.885} C_VEL
LIN {X 0,Y 200.139,Z 380.555,A -85,B 0,C 180,E1 -21411.926,E2 -21411.926} C_VEL
LIN {X 0,Y 200.328,Z 380.519,A -85,B 0,C 180,E1 -21417.99,E2 -21417.99} C_VEL
LIN {X 0,Y 200.486,Z 380.503,A -85,B 0,C 180,E1 -21420,E2 -21420} C_VEL
LIN {X 0,Y 200.038,Z 380.566,A -85,B 0,C 180,E1 -21424.03,E2 -21424.03} C_VEL
LIN {X 0,Y 200.131,Z 380.545,A -85,B 0,C 180,E1 -21428.075,E2 -21428.075} C_VEL
LIN {X 0,Y 199.921,Z 380.58,A -85,B 0,C 180,E1 -21432.177,E2 -21432.177} C_VEL
LIN {X 0,Y 199.811,Z 380.587,A -85,B 0,C 180,E1 -21436.343,E2 -21436.343} C_VEL
LIN {X 0,Y 199.707,Z 380.605,A -85,B 0,C 180,E1 -21440.605,E2 -21440.605} C_VEL
LIN {X 0,Y 199.68,Z 380.608,A -85,B 0,C 180,E1 -21444.984,E2 -21444.984} C_VEL
LIN {X 0,Y 199.681,Z 380.604,A -85,B 0,C 180,E1 -21449.522,E2 -21449.522} C_VEL
LIN {X 0,Y 199.671,Z 380.611,A -85,B 0,C 180,E1 -21452.352,E2 -21452.352} C_VEL
LIN {X 0,Y 199.646,Z 380.615,A -85,B 0,C 180,E1 -21456.759,E2 -21456.759} C_VEL
LIN {X 0,Y 199.645,Z 380.614,A -85,B 0,C 180,E1 -21459.32,E2 -21459.32} C_VEL
LIN {X 0,Y 199.588,Z 380.619,A -85,B 0,C 180,E1 -21464.77,E2 -21464.77} C_VEL
LIN {X 0,Y 199.586,Z 380.62,A -85,B 0,C 180,E1 -21468.005,E2 -21468.005} C_VEL
LIN {X 0,Y 199.617,Z 380.617,A -85,B 0,C 180,E1 -21470.767,E2 -21470.767} C_VEL
LIN {X 0,Y 199.619,Z 380.619,A -85,B 0,C 180,E1 -21475.713,E2 -21475.713} C_VEL
LIN {X 0,Y 199.707,Z 380.608,A -85,B 0,C 180,E1 -21478.136,E2 -21478.136} C_VEL
LIN {X 0,Y 199.693,Z 380.611,A -85,B 0,C 180,E1 -21482.771,E2 -21482.771} C_VEL
LIN {X 0,Y 199.708,Z 380.608,A -85,B 0,C 180,E1 -21485.625,E2 -21485.625} C_VEL
LIN {X 0,Y 200.841,Z 383.61,A -85,B 0,C 180,E1 -21486.106,E2 -21486.106} C_VEL
LIN {X 0,Y 205.533,Z 394.65,A -85,B 0,C 180,E1 -21488.144,E2 -21488.144} C_VEL
LIN {X 0,Y 209.123,Z 404.938,A -85,B 0,C 180,E1 -21490.222,E2 -21490.222} C_VEL
LIN {X 0,Y 211.54,Z 414.445,A -85,B 0,C 180,E1 -21492.305,E2 -21492.305} C_VEL
LIN {X 0,Y 209.48,Z 425.119,A -85,B 0,C 180,E1 -21494.43,E2 -21494.43} C_VEL
LIN {X 0,Y 207.506,Z 434.528,A -85,B 0,C 180,E1 -21496.783,E2 -21496.783} C_VEL
LIN {X 0,Y 205.634,Z 442.27,A -85,B 0,C 180,E1 -21499.164,E2 -21499.164} C_VEL
LIN {X 0,Y 203.677,Z 449.848,A -85,B 0,C 180,E1 -21502.065,E2 -21502.065} C_VEL
LIN {X 0,Y 202.179,Z 455.927,A -85,B 0,C 180,E1 -21505.013,E2 -21505.013} C_VEL
LIN {X 0,Y 201.03,Z 460.768,A -85,B 0,C 180,E1 -21507.995,E2 -21507.995} C_VEL
LIN {X 0,Y 200.056,Z 464.542,A -85,B 0,C 180,E1 -21511.005,E2 -21511.005} C_VEL
LIN {X 0,Y 199.614,Z 467.293,A -85,B 0,C 180,E1 -21514.036,E2 -21514.036} C_VEL
LIN {X 0,Y 199.622,Z 468.588,A -85,B 0,C 180,E1 -21516.061,E2 -21516.061} C_VEL
LIN {X 0,Y 199.793,Z 470.024,A -85,B 0,C 180,E1 -21519.952,E2 -21519.952} C_VEL
LIN {X 0,Y 200.118,Z 470.167,A -85,B 0,C 180,E1 -21522.163,E2 -21522.163} C_VEL
LIN {X 0,Y 201.242,Z 469.268,A -85,B 0,C 180,E1 -21526.222,E2 -21526.222} C_VEL
LIN {X 0,Y 202.075,Z 468.203,A -85,B 0,C 180,E1 -21528.239,E2 -21528.239} C_VEL
LIN {X 0,Y 203.918,Z 465.56,A -85,B 0,C 180,E1 -21531.477,E2 -21531.477} C_VEL
LIN {X 0,Y 206.519,Z 461.035,A -85,B 0,C 180,E1 -21535.173,E2 -21535.173} C_VEL
LIN {X 0,Y 209.04,Z 456.133,A -85,B 0,C 180,E1 -21538.077,E2 -21538.077} C_VEL
LIN {X 0,Y 211.952,Z 450.129,A -85,B 0,C 180,E1 -21540.815,E2 -21540.815} C_VEL
LIN {X 0,Y 215.436,Z 442.016,A -85,B 0,C 180,E1 -21543.68,E2 -21543.68} C_VEL
LIN {X 0,Y 218.778,Z 433.194,A -85,B 0,C 180,E1 -21546.125,E2 -21546.125} C_VEL
LIN {X 0,Y 219.936,Z 429.625,A -85,B 0,C 180,E1 -21546.977,E2 -21546.977} C_VEL
LIN {X 0,Y 218.373,Z 421.896,A -85,B 0,C 180,E1 -21549.429,E2 -21549.429} C_VEL
LIN {X 0,Y 215.688,Z 412.884,A -85,B 0,C 180,E1 -21552.158,E2 -21552.158} C_VEL
LIN {X 0,Y 211.684,Z 402.886,A -85,B 0,C 180,E1 -21555.128,E2 -21555.128} C_VEL
LIN {X 0,Y 207.049,Z 393.577,A -85,B 0,C 180,E1 -21557.903,E2 -21557.903} C_VEL
LIN {X 0,Y 202.639,Z 385.969,A -85,B 0,C 180,E1 -21560.225,E2 -21560.225} C_VEL
LIN {X 0,Y 201.804,Z 384.83,A -85,B 0,C 180,E1 -21560.627,E2 -21560.627} C_VEL
LIN {X 0,Y 200.207,Z 382.456,A -85,B 0,C 180,E1 -21561.404,E2 -21561.404} C_VEL
LIN {X 0,Y 199.713,Z 380.612,A -85,B 0,C 180,E1 -21561.826,E2 -21561.826} C_VEL
LIN {X 0,Y 199.633,Z 380.62,A -85,B 0,C 180,E1 -21565.717,E2 -21565.717} C_VEL
LIN {X 0,Y 199.694,Z 380.571,A -85,B 0,C 180,E1 -21568.135,E2 -21568.135} C_VEL
LIN {X 0,Y 199.683,Z 380.59,A -85,B 0,C 180,E1 -21572.771,E2 -21572.771} C_VEL
LIN {X 0,Y 199.735,Z 380.589,A -85,B 0,C 180,E1 -21577.228,E2 -21577.228} C_VEL
LIN {X 0,Y 199.793,Z 380.583,A -85,B 0,C 180,E1 -21581.757,E2 -21581.757} C_VEL
LIN {X 0,Y 199.845,Z 380.591,A -85,B 0,C 180,E1 -21585.748,E2 -21585.748} C_VEL
LIN {X 0,Y 200.072,Z 380.559,A -85,B 0,C 180,E1 -21589.884,E2 -21589.884} C_VEL
LIN {X 0,Y 200.038,Z 380.549,A -85,B 0,C 180,E1 -21593.949,E2 -21593.949} C_VEL
LIN {X 0,Y 200.322,Z 380.529,A -85,B 0,C 180,E1 -21597.989,E2 -21597.989} C_VEL
LIN {X 0,Y 200.48,Z 380.496,A -85,B 0,C 180,E1 -21600,E2 -21600} C_VEL
LIN {X 0,Y 200.032,Z 380.559,A -85,B 0,C 180,E1 -21604.029,E2 -21604.029} C_VEL
LIN {X 0,Y 200.128,Z 380.555,A -85,B 0,C 180,E1 -21608.075,E2 -21608.075} C_VEL
LIN {X 0,Y 199.911,Z 380.582,A -85,B 0,C 180,E1 -21612.177,E2 -21612.177} C_VEL
LIN {X 0,Y 199.802,Z 380.595,A -85,B 0,C 180,E1 -21616.343,E2 -21616.343} C_VEL
LIN {X 0,Y 199.82,Z 380.59,A -85,B 0,C 180,E1 -21618.454,E2 -21618.454} C_VEL
LIN {X 0,Y 199.743,Z 380.769,A -85,B 0,C 180,E1 -21622.497,E2 -21622.497} C_VEL
LIN {X 0,Y 200.478,Z 384.288,A -85,B 0,C 180,E1 -21627.112,E2 -21627.112} C_VEL
LIN {X 0,Y 201.267,Z 388.154,A -85,B 0,C 180,E1 -21631.586,E2 -21631.586} C_VEL
LIN {X 0,Y 202.267,Z 392.608,A -85,B 0,C 180,E1 -21636.205,E2 -21636.205} C_VEL
LIN {X 0,Y 203.203,Z 397.799,A -85,B 0,C 180,E1 -21641.081,E2 -21641.081} C_VEL
LIN {X 0,Y 204.018,Z 402.222,A -85,B 0,C 180,E1 -21644.925,E2 -21644.925} C_VEL
LIN {X 0,Y 204.443,Z 404.707,A -85,B 0,C 180,E1 -21646.979,E2 -21646.979} C_VEL
LIN {X 0,Y 205.72,Z 408.306,A -85,B 0,C 180,E1 -21647.564,E2 -21647.564} C_VEL
LIN {X 0,Y 207.351,Z 411.126,A -85,B 0,C 180,E1 -21648.217,E2 -21648.217} C_VEL
LIN {X 0,Y 209.038,Z 415.865,A -85,B 0,C 180,E1 -21649.035,E2 -21649.035} C_VEL
LIN {X 0,Y 211.463,Z 427.837,A -85,B 0,C 180,E1 -21650.843,E2 -21650.843} C_VEL
LIN {X 0,Y 212.957,Z 440.143,A -85,B 0,C 180,E1 -21652.817,E2 -21652.817} C_VEL
LIN {X 0,Y 213.46,Z 450.456,A -85,B 0,C 180,E1 -21654.618,E2 -21654.618} C_VEL
LIN {X 0,Y 213.265,Z 461.566,A -85,B 0,C 180,E1 -21656.781,E2 -21656.781} C_VEL
LIN {X 0,Y 212.304,Z 471.939,A -85,B 0,C 180,E1 -21659.077,E2 -21659.077} C_VEL
LIN {X 0,Y 210.624,Z 481.781,A -85,B 0,C 180,E1 -21661.611,E2 -21661.611} C_VEL
LIN {X 0,Y 208.83,Z 488.208,A -85,B 0,C 180,E1 -21663.52,E2 -21663.52} C_VEL
LIN {X 0,Y 205.47,Z 496.276,A -85,B 0,C 180,E1 -21666.304,E2 -21666.304} C_VEL
LIN {X 0,Y 202.474,Z 503.543,A -85,B 0,C 180,E1 -21669.584,E2 -21669.584} C_VEL
LIN {X 0,Y 200.412,Z 508.794,A -85,B 0,C 180,E1 -21672.66,E2 -21672.66} C_VEL
LIN {X 0,Y 200.025,Z 509.89,A -85,B 0,C 180,E1 -21673.415,E2 -21673.415} C_VEL
LIN {X 0,Y 198.668,Z 511.935,A -85,B 0,C 180,E1 -21674.959,E2 -21674.959} C_VEL
LIN {X 0,Y 194.971,Z 514.514,A -85,B 0,C 180,E1 -21677.531,E2 -21677.531} C_VEL
LIN {X 0,Y 191.705,Z 516.328,A -85,B 0,C 180,E1 -21680.257,E2 -21680.257} C_VEL
LIN {X 0,Y 191.053,Z 517.16,A -85,B 0,C 180,E1 -21681.999,E2 -21681.999} C_VEL
LIN {X 0,Y 191.531,Z 518.252,A -85,B 0,C 180,E1 -21685.793,E2 -21685.793} C_VEL
LIN {X 0,Y 191.867,Z 518.292,A -85,B 0,C 180,E1 -21687.902,E2 -21687.902} C_VEL
LIN {X 0,Y 192.044,Z 517.855,A -85,B 0,C 180,E1 -21690.002,E2 -21690.002} C_VEL
LIN {X 0,Y 191.948,Z 516.951,A -85,B 0,C 180,E1 -21692.1,E2 -21692.1} C_VEL
LIN {X 0,Y 191.656,Z 515.594,A -85,B 0,C 180,E1 -21694.207,E2 -21694.207} C_VEL
LIN {X 0,Y 191.299,Z 512.791,A -85,B 0,C 180,E1 -21697.283,E2 -21697.283} C_VEL
LIN {X 0,Y 191.303,Z 508.695,A -85,B 0,C 180,E1 -21700.586,E2 -21700.586} C_VEL
LIN {X 0,Y 192.005,Z 502.603,A -85,B 0,C 180,E1 -21704.306,E2 -21704.306} C_VEL
LIN {X 0,Y 193.133,Z 495.878,A -85,B 0,C 180,E1 -21707.472,E2 -21707.472} C_VEL
LIN {X 0,Y 195.138,Z 487.638,A -85,B 0,C 180,E1 -21710.544,E2 -21710.544} C_VEL
LIN {X 0,Y 196.573,Z 480.922,A -85,B 0,C 180,E1 -21712.604,E2 -21712.604} C_VEL
LIN {X 0,Y 197.428,Z 470.65,A -85,B 0,C 180,E1 -21715.29,E2 -21715.29} C_VEL
LIN {X 0,Y 198.302,Z 459.662,A -85,B 0,C 180,E1 -21717.622,E2 -21717.622} C_VEL
LIN {X 0,Y 198.603,Z 447.682,A -85,B 0,C 180,E1 -21719.699,E2 -21719.699} C_VEL
LIN {X 0,Y 198.187,Z 435.212,A -85,B 0,C 180,E1 -21721.485,E2 -21721.485} C_VEL
LIN {X 0,Y 196.825,Z 421.725,A -85,B 0,C 180,E1 -21723.078,E2 -21723.078} C_VEL
LIN {X 0,Y 194.338,Z 407.387,A -85,B 0,C 180,E1 -21724.47,E2 -21724.47} C_VEL
LIN {X 0,Y 195.948,Z 401.191,A -85,B 0,C 180,E1 -21728.879,E2 -21728.879} C_VEL
LIN {X 0,Y 195.827,Z 398.241,A -85,B 0,C 180,E1 -21731.091,E2 -21731.091} C_VEL
LIN {X 0,Y 194.897,Z 393.096,A -85,B 0,C 180,E1 -21735.219,E2 -21735.219} C_VEL
LIN {X 0,Y 193.878,Z 387.971,A -85,B 0,C 180,E1 -21739.576,E2 -21739.576} C_VEL
LIN {X 0,Y 192.872,Z 382.787,A -85,B 0,C 180,E1 -21744.337,E2 -21744.337} C_VEL
LIN {X 0,Y 192.606,Z 381.497,A -85,B 0,C 180,E1 -21745.716,E2 -21745.716} C_VEL
LIN {X 0,Y 192.649,Z 381.489,A -85,B 0,C 180,E1 -21751.112,E2 -21751.112} C_VEL
LIN {X 0,Y 192.711,Z 381.484,A -85,B 0,C 180,E1 -21756.35,E2 -21756.35} C_VEL
LIN {X 0,Y 192.787,Z 381.474,A -85,B 0,C 180,E1 -21761.415,E2 -21761.415} C_VEL
LIN {X 0,Y 192.859,Z 381.461,A -85,B 0,C 180,E1 -21767.371,E2 -21767.371} C_VEL
LIN {X 0,Y 193.085,Z 381.433,A -85,B 0,C 180,E1 -21771.629,E2 -21771.629} C_VEL
LIN {X 0,Y 193.27,Z 381.398,A -85,B 0,C 180,E1 -21777.917,E2 -21777.917} C_VEL
LIN {X 0,Y 193.45,Z 381.379,A -85,B 0,C 180,E1 -21780,E2 -21780} C_VEL
LIN {X 0,Y 192.984,Z 381.443,A -85,B 0,C 180,E1 -21784.177,E2 -21784.177} C_VEL
LIN {X 0,Y 193.079,Z 381.425,A -85,B 0,C 180,E1 -21788.372,E2 -21788.372} C_VEL
LIN {X 0,Y 192.86,Z 381.457,A -85,B 0,C 180,E1 -21792.63,E2 -21792.63} C_VEL
LIN {X 0,Y 192.764,Z 381.467,A -85,B 0,C 180,E1 -21796.959,E2 -21796.959} C_VEL
LIN {X 0,Y 192.644,Z 381.483,A -85,B 0,C 180,E1 -21801.397,E2 -21801.397} C_VEL
LIN {X 0,Y 192.671,Z 381.478,A -85,B 0,C 180,E1 -21804.225,E2 -21804.225} C_VEL
LIN {X 0,Y 192.656,Z 381.483,A -85,B 0,C 180,E1 -21808.892,E2 -21808.892} C_VEL
LIN {X 0,Y 192.607,Z 381.492,A -85,B 0,C 180,E1 -21813.185,E2 -21813.185} C_VEL
LIN {X 0,Y 192.616,Z 381.49,A -85,B 0,C 180,E1 -21816.607,E2 -21816.607} C_VEL
LIN {X 0,Y 192.53,Z 381.501,A -85,B 0,C 180,E1 -21821.077,E2 -21821.077} C_VEL
LIN {X 0,Y 192.499,Z 381.503,A -85,B 0,C 180,E1 -21826.076,E2 -21826.076} C_VEL
LIN {X 0,Y 192.524,Z 381.499,A -85,B 0,C 180,E1 -21830.05,E2 -21830.05} C_VEL
LIN {X 0,Y 192.566,Z 381.496,A -85,B 0,C 180,E1 -21834.27,E2 -21834.27} C_VEL
LIN {X 0,Y 192.616,Z 381.491,A -85,B 0,C 180,E1 -21837.057,E2 -21837.057} C_VEL
LIN {X 0,Y 192.671,Z 381.486,A -85,B 0,C 180,E1 -21841.691,E2 -21841.691} C_VEL
LIN {X 0,Y 192.64,Z 381.595,A -85,B 0,C 180,E1 -21844.458,E2 -21844.458} C_VEL
LIN {X 0,Y 193.743,Z 384.491,A -85,B 0,C 180,E1 -21844.953,E2 -21844.953} C_VEL
LIN {X 0,Y 198.554,Z 395.206,A -85,B 0,C 180,E1 -21847.084,E2 -21847.084} C_VEL
LIN {X 0,Y 202.094,Z 405.271,A -85,B 0,C 180,E1 -21849.206,E2 -21849.206} C_VEL
LIN {X 0,Y 204.641,Z 414.692,A -85,B 0,C 180,E1 -21851.367,E2 -21851.367} C_VEL
LIN {X 0,Y 204.871,Z 416.094,A -85,B 0,C 180,E1 -21851.702,E2 -21851.702} C_VEL
LIN {X 0,Y 202.739,Z 426.659,A -85,B 0,C 180,E1 -21853.898,E2 -21853.898} C_VEL
LIN {X 0,Y 200.665,Z 435.951,A -85,B 0,C 180,E1 -21856.324,E2 -21856.324} C_VEL
LIN {X 0,Y 198.385,Z 444.921,A -85,B 0,C 180,E1 -21859.28,E2 -21859.28} C_VEL
LIN {X 0,Y 196.442,Z 452.166,A -85,B 0,C 180,E1 -21862.288,E2 -21862.288} C_VEL
LIN {X 0,Y 195.175,Z 457.079,A -85,B 0,C 180,E1 -21864.834,E2 -21864.834} C_VEL
LIN {X 0,Y 193.98,Z 461.863,A -85,B 0,C 180,E1 -21867.922,E2 -21867.922} C_VEL
LIN {X 0,Y 192.984,Z 465.584,A -85,B 0,C 180,E1 -21871.042,E2 -21871.042} C_VEL
LIN {X 0,Y 192.561,Z 468.28,A -85,B 0,C 180,E1 -21874.185,E2 -21874.185} C_VEL
LIN {X 0,Y 192.567,Z 469.553,A -85,B 0,C 180,E1 -21876.284,E2 -21876.284} C_VEL
LIN {X 0,Y 192.78,Z 470.899,A -85,B 0,C 180,E1 -21880.156,E2 -21880.156} C_VEL
LIN {X 0,Y 193.151,Z 471.035,A -85,B 0,C 180,E1 -21882.609,E2 -21882.609} C_VEL
LIN {X 0,Y 194.408,Z 470.081,A -85,B 0,C 180,E1 -21886.809,E2 -21886.809} C_VEL
LIN {X 0,Y 195.301,Z 468.969,A -85,B 0,C 180,E1 -21888.895,E2 -21888.895} C_VEL
LIN {X 0,Y 197.153,Z 466.461,A -85,B 0,C 180,E1 -21892.051,E2 -21892.051} C_VEL
LIN {X 0,Y 199.249,Z 463.081,A -85,B 0,C 180,E1 -21895.04,E2 -21895.04} C_VEL
LIN {X 0,Y 201.822,Z 458.501,A -85,B 0,C 180,E1 -21898.04,E2 -21898.04} C_VEL
LIN {X 0,Y 204.823,Z 452.644,A -85,B 0,C 180,E1 -21900.975,E2 -21900.975} C_VEL
LIN {X 0,Y 208.307,Z 445.282,A -85,B 0,C 180,E1 -21903.825,E2 -21903.825} C_VEL
LIN {X 0,Y 211.456,Z 437.719,A -85,B 0,C 180,E1 -21906.151,E2 -21906.151} C_VEL
LIN {X 0,Y 213.454,Z 432.288,A -85,B 0,C 180,E1 -21907.559,E2 -21907.559} C_VEL
LIN {X 0,Y 213.323,Z 429.928,A -85,B 0,C 180,E1 -21908.324,E2 -21908.324} C_VEL
LIN {X 0,Y 211.518,Z 421.654,A -85,B 0,C 180,E1 -21911.084,E2 -21911.084} C_VEL
LIN {X 0,Y 208.98,Z 413.583,A -85,B 0,C 180,E1 -21913.677,E2 -21913.677} C_VEL
LIN {X 0,Y 205.063,Z 404.024,A -85,B 0,C 180,E1 -21916.728,E2 -21916.728} C_VEL
LIN {X 0,Y 200.622,Z 395.104,A -85,B 0,C 180,E1 -21919.603,E2 -21919.603} C_VEL
LIN {X 0,Y 198.244,Z 390.845,A -85,B 0,C 180,E1 -21921.004,E2 -21921.004} C_VEL
LIN {X 0,Y 196.117,Z 387.756,A -85,B 0,C 180,E1 -21922.142,E2 -21922.142} C_VEL
LIN {X 0,Y 195.349,Z 386.235,A -85,B 0,C 180,E1 -21922.609,E2 -21922.609} C_VEL
LIN {X 0,Y 193.367,Z 383.898,A -85,B 0,C 180,E1 -21923.604,E2 -21923.604} C_VEL
LIN {X 0,Y 192.604,Z 381.487,A -85,B 0,C 180,E1 -21924.19,E2 -21924.19} C_VEL
LIN {X 0,Y 192.597,Z 381.443,A -85,B 0,C 180,E1 -21929.277,E2 -21929.277} C_VEL
LIN {X 0,Y 192.658,Z 381.445,A -85,B 0,C 180,E1 -21931.69,E2 -21931.69} C_VEL
LIN {X 0,Y 192.703,Z 381.466,A -85,B 0,C 180,E1 -21936.348,E2 -21936.348} C_VEL
LIN {X 0,Y 192.729,Z 381.464,A -85,B 0,C 180,E1 -21941.456,E2 -21941.456} C_VEL
LIN {X 0,Y 192.769,Z 381.474,A -85,B 0,C 180,E1 -21945.214,E2 -21945.214} C_VEL
LIN {X 0,Y 193.017,Z 381.438,A -85,B 0,C 180,E1 -21949.51,E2 -21949.51} C_VEL
LIN {X 0,Y 193.002,Z 381.426,A -85,B 0,C 180,E1 -21953.728,E2 -21953.728} C_VEL
LIN {X 0,Y 193.263,Z 381.409,A -85,B 0,C 180,E1 -21957.916,E2 -21957.916} C_VEL
LIN {X 0,Y 193.444,Z 381.372,A -85,B 0,C 180,E1 -21960,E2 -21960} C_VEL
LIN {X 0,Y 192.978,Z 381.436,A -85,B 0,C 180,E1 -21964.177,E2 -21964.177} C_VEL
LIN {X 0,Y 193.075,Z 381.43,A -85,B 0,C 180,E1 -21968.372,E2 -21968.372} C_VEL
LIN {X 0,Y 192.849,Z 381.458,A -85,B 0,C 180,E1 -21972.63,E2 -21972.63} C_VEL
LIN {X 0,Y 192.777,Z 381.467,A -85,B 0,C 180,E1 -21978.586,E2 -21978.586} C_VEL
LIN {X 0,Y 192.686,Z 381.572,A -85,B 0,C 180,E1 -21980.552,E2 -21980.552} C_VEL
LIN {X 0,Y 193.268,Z 384.422,A -85,B 0,C 180,E1 -21984.623,E2 -21984.623} C_VEL
LIN {X 0,Y 194.103,Z 388.397,A -85,B 0,C 180,E1 -21989.662,E2 -21989.662} C_VEL
LIN {X 0,Y 195.172,Z 393.394,A -85,B 0,C 180,E1 -21995.18,E2 -21995.18} C_VEL
LIN {X 0,Y 196.128,Z 398.463,A -85,B 0,C 180,E1 -22000.166,E2 -22000.166} C_VEL
LIN {X 0,Y 197.038,Z 403.399,A -85,B 0,C 180,E1 -22004.654,E2 -22004.654} C_VEL
LIN {X 0,Y 198.344,Z 406.991,A -85,B 0,C 180,E1 -22005.305,E2 -22005.305} C_VEL
LIN {X 0,Y 200.226,Z 410.075,A -85,B 0,C 180,E1 -22006.126,E2 -22006.126} C_VEL
LIN {X 0,Y 202.135,Z 414.392,A -85,B 0,C 180,E1 -22007.05,E2 -22007.05} C_VEL
LIN {X 0,Y 203.894,Z 418.855,A -85,B 0,C 180,E1 -22007.961,E2 -22007.961} C_VEL
LIN {X 0,Y 206.124,Z 431.878,A -85,B 0,C 180,E1 -22010.098,E2 -22010.098} C_VEL
LIN {X 0,Y 207.182,Z 443.986,A -85,B 0,C 180,E1 -22012.215,E2 -22012.215} C_VEL
LIN {X 0,Y 207.274,Z 455.709,A -85,B 0,C 180,E1 -22014.465,E2 -22014.465} C_VEL
LIN {X 0,Y 206.582,Z 466.253,A -85,B 0,C 180,E1 -22016.743,E2 -22016.743} C_VEL
LIN {X 0,Y 205.302,Z 475.8,A -85,B 0,C 180,E1 -22019.105,E2 -22019.105} C_VEL
LIN {X 0,Y 203.402,Z 484.627,A -85,B 0,C 180,E1 -22021.636,E2 -22021.636} C_VEL
LIN {X 0,Y 200.66,Z 491.905,A -85,B 0,C 180,E1 -22024.038,E2 -22024.038} C_VEL
LIN {X 0,Y 197.445,Z 499.074,A -85,B 0,C 180,E1 -22026.951,E2 -22026.951} C_VEL
LIN {X 0,Y 194.652,Z 505.446,A -85,B 0,C 180,E1 -22030.315,E2 -22030.315} C_VEL
LIN {X 0,Y 192.555,Z 510.832,A -85,B 0,C 180,E1 -22034.115,E2 -22034.115} C_VEL
LIN {X 0,Y 191.456,Z 514.076,A -85,B 0,C 180,E1 -22037.278,E2 -22037.278} C_VEL
LIN {X 0,Y 191.12,Z 515.739,A -85,B 0,C 180,E1 -22039.407,E2 -22039.407} C_VEL
LIN {X 0,Y 191.053,Z 517.16,A -85,B 0,C 180,E1 -22041.999,E2 -22041.999} C_VEL
LIN {X 0,Y 190.556,Z 517.773,A -85,B 0,C 180,E1 -22043.759,E2 -22043.759} C_VEL
LIN {X 0,Y 189.208,Z 517.955,A -85,B 0,C 180,E1 -22045.507,E2 -22045.507} C_VEL
LIN {X 0,Y 185.929,Z 517.314,A -85,B 0,C 180,E1 -22049.045,E2 -22049.045} C_VEL
LIN {X 0,Y 184.895,Z 516.302,A -85,B 0,C 180,E1 -22051.491,E2 -22051.491} C_VEL
LIN {X 0,Y 184.565,Z 514.626,A -85,B 0,C 180,E1 -22054.369,E2 -22054.369} C_VEL
LIN {X 0,Y 184.226,Z 512.031,A -85,B 0,C 180,E1 -22057.313,E2 -22057.313} C_VEL
LIN {X 0,Y 184.266,Z 507.633,A -85,B 0,C 180,E1 -22060.995,E2 -22060.995} C_VEL
LIN {X 0,Y 185.058,Z 501.466,A -85,B 0,C 180,E1 -22064.855,E2 -22064.855} C_VEL
LIN {X 0,Y 186.307,Z 494.685,A -85,B 0,C 180,E1 -22068.134,E2 -22068.134} C_VEL
LIN {X 0,Y 188.578,Z 485.947,A -85,B 0,C 180,E1 -22071.459,E2 -22071.459} C_VEL
LIN {X 0,Y 189.796,Z 479.556,A -85,B 0,C 180,E1 -22073.459,E2 -22073.459} C_VEL
LIN {X 0,Y 190.745,Z 469.182,A -85,B 0,C 180,E1 -22076.242,E2 -22076.242} C_VEL
LIN {X 0,Y 191.586,Z 458.949,A -85,B 0,C 180,E1 -22078.484,E2 -22078.484} C_VEL
LIN {X 0,Y 191.936,Z 447.665,A -85,B 0,C 180,E1 -22080.536,E2 -22080.536} C_VEL
LIN {X 0,Y 191.687,Z 436.015,A -85,B 0,C 180,E1 -22082.299,E2 -22082.299} C_VEL
LIN {X 0,Y 190.475,Z 422.958,A -85,B 0,C 180,E1 -22083.963,E2 -22083.963} C_VEL
LIN {X 0,Y 188.211,Z 409.62,A -85,B 0,C 180,E1 -22085.392,E2 -22085.392} C_VEL
LIN {X 0,Y 187.689,Z 406.457,A -85,B 0,C 180,E1 -22085.684,E2 -22085.684} C_VEL
LIN {X 0,Y 188.923,Z 401.71,A -85,B 0,C 180,E1 -22089.23,E2 -22089.23} C_VEL
LIN {X 0,Y 188.617,Z 398.062,A -85,B 0,C 180,E1 -22092.123,E2 -22092.123} C_VEL
LIN {X 0,Y 187.606,Z 392.958,A -85,B 0,C 180,E1 -22096.412,E2 -22096.412} C_VEL
LIN {X 0,Y 186.561,Z 387.409,A -85,B 0,C 180,E1 -22101.455,E2 -22101.455} C_VEL
LIN {X 0,Y 185.566,Z 382.373,A -85,B 0,C 180,E1 -22106.433,E2 -22106.433} C_VEL
LIN {X 0,Y 185.585,Z 382.369,A -85,B 0,C 180,E1 -22110.578,E2 -22110.578} C_VEL
LIN {X 0,Y 185.593,Z 382.37,A -85,B 0,C 180,E1 -22115.384,E2 -22115.384} C_VEL
LIN {X 0,Y 185.7,Z 382.358,A -85,B 0,C 180,E1 -22121.116,E2 -22121.116} C_VEL
LIN {X 0,Y 185.734,Z 382.352,A -85,B 0,C 180,E1 -22124.641,E2 -22124.641} C_VEL
LIN {X 0,Y 185.949,Z 382.322,A -85,B 0,C 180,E1 -22129.329,E2 -22129.329} C_VEL
LIN {X 0,Y 185.975,Z 382.318,A -85,B 0,C 180,E1 -22133.491,E2 -22133.491} C_VEL
LIN {X 0,Y 186.214,Z 382.276,A -85,B 0,C 180,E1 -22137.838,E2 -22137.838} C_VEL
LIN {X 0,Y 186.413,Z 382.255,A -85,B 0,C 180,E1 -22140,E2 -22140} C_VEL
LIN {X 0,Y 185.932,Z 382.32,A -85,B 0,C 180,E1 -22144.336,E2 -22144.336} C_VEL
LIN {X 0,Y 186.031,Z 382.305,A -85,B 0,C 180,E1 -22148.692,E2 -22148.692} C_VEL
LIN {X 0,Y 185.772,Z 382.34,A -85,B 0,C 180,E1 -22153.12,E2 -22153.12} C_VEL
LIN {X 0,Y 185.681,Z 382.354,A -85,B 0,C 180,E1 -22158.867,E2 -22158.867} C_VEL
LIN {X 0,Y 185.604,Z 382.353,A -85,B 0,C 180,E1 -22162.251,E2 -22162.251} C_VEL
LIN {X 0,Y 185.569,Z 382.369,A -85,B 0,C 180,E1 -22167.032,E2 -22167.032} C_VEL
LIN {X 0,Y 185.585,Z 382.359,A -85,B 0,C 180,E1 -22169.493,E2 -22169.493} C_VEL
LIN {X 0,Y 185.525,Z 382.374,A -85,B 0,C 180,E1 -22174.627,E2 -22174.627} C_VEL
LIN {X 0,Y 185.55,Z 382.373,A -85,B 0,C 180,E1 -22177.304,E2 -22177.304} C_VEL
LIN {X 0,Y 185.492,Z 382.377,A -85,B 0,C 180,E1 -22180.73,E2 -22180.73} C_VEL
LIN {X 0,Y 185.488,Z 382.376,A -85,B 0,C 180,E1 -22183.952,E2 -22183.952} C_VEL
LIN {X 0,Y 185.477,Z 382.378,A -85,B 0,C 180,E1 -22189.274,E2 -22189.274} C_VEL
LIN {X 0,Y 185.512,Z 382.373,A -85,B 0,C 180,E1 -22192.711,E2 -22192.711} C_VEL
LIN {X 0,Y 185.552,Z 382.371,A -85,B 0,C 180,E1 -22197.975,E2 -22197.975} C_VEL
LIN {X 0,Y 185.588,Z 382.368,A -85,B 0,C 180,E1 -22200.575,E2 -22200.575} C_VEL
LIN {X 0,Y 185.555,Z 382.372,A -85,B 0,C 180,E1 -22203.125,E2 -22203.125} C_VEL
LIN {X 0,Y 186.619,Z 385.312,A -85,B 0,C 180,E1 -22203.685,E2 -22203.685} C_VEL
LIN {X 0,Y 191.233,Z 395.208,A -85,B 0,C 180,E1 -22205.801,E2 -22205.801} C_VEL
LIN {X 0,Y 195.183,Z 406.06,A -85,B 0,C 180,E1 -22208.214,E2 -22208.214} C_VEL
LIN {X 0,Y 197.667,Z 414.913,A -85,B 0,C 180,E1 -22210.345,E2 -22210.345} C_VEL
LIN {X 0,Y 198.257,Z 417.75,A -85,B 0,C 180,E1 -22211.065,E2 -22211.065} C_VEL
LIN {X 0,Y 196.048,Z 428.191,A -85,B 0,C 180,E1 -22213.333,E2 -22213.333} C_VEL
LIN {X 0,Y 193.868,Z 437.336,A -85,B 0,C 180,E1 -22215.834,E2 -22215.834} C_VEL
LIN {X 0,Y 191.483,Z 446.216,A -85,B 0,C 180,E1 -22218.889,E2 -22218.889} C_VEL
LIN {X 0,Y 189.474,Z 453.387,A -85,B 0,C 180,E1 -22222.003,E2 -22222.003} C_VEL
LIN {X 0,Y 188.172,Z 458.233,A -85,B 0,C 180,E1 -22224.641,E2 -22224.641} C_VEL
LIN {X 0,Y 186.932,Z 462.959,A -85,B 0,C 180,E1 -22227.844,E2 -22227.844} C_VEL
LIN {X 0,Y 185.916,Z 466.625,A -85,B 0,C 180,E1 -22231.081,E2 -22231.081} C_VEL
LIN {X 0,Y 185.509,Z 469.268,A -85,B 0,C 180,E1 -22234.344,E2 -22234.344} C_VEL
LIN {X 0,Y 185.518,Z 470.518,A -85,B 0,C 180,E1 -22236.524,E2 -22236.524} C_VEL
LIN {X 0,Y 185.776,Z 471.775,A -85,B 0,C 180,E1 -22240.389,E2 -22240.389} C_VEL
LIN {X 0,Y 186.206,Z 471.902,A -85,B 0,C 180,E1 -22243.087,E2 -22243.087} C_VEL
LIN {X 0,Y 186.804,Z 471.592,A -85,B 0,C 180,E1 -22245.268,E2 -22245.268} C_VEL
LIN {X 0,Y 187.576,Z 470.882,A -85,B 0,C 180,E1 -22247.44,E2 -22247.44} C_VEL
LIN {X 0,Y 188.557,Z 469.734,A -85,B 0,C 180,E1 -22249.598,E2 -22249.598} C_VEL
LIN {X 0,Y 190.438,Z 467.339,A -85,B 0,C 180,E1 -22252.687,E2 -22252.687} C_VEL
LIN {X 0,Y 192.776,Z 463.737,A -85,B 0,C 180,E1 -22255.942,E2 -22255.942} C_VEL
LIN {X 0,Y 195.506,Z 459.097,A -85,B 0,C 180,E1 -22259.03,E2 -22259.03} C_VEL
LIN {X 0,Y 198.723,Z 453.17,A -85,B 0,C 180,E1 -22262.037,E2 -22262.037} C_VEL
LIN {X 0,Y 202.378,Z 445.735,A -85,B 0,C 180,E1 -22264.958,E2 -22264.958} C_VEL
LIN {X 0,Y 205.706,Z 438.083,A -85,B 0,C 180,E1 -22267.33,E2 -22267.33} C_VEL
LIN {X 0,Y 207.259,Z 433.812,A -85,B 0,C 180,E1 -22268.485,E2 -22268.485} C_VEL
LIN {X 0,Y 205.825,Z 425.975,A -85,B 0,C 180,E1 -22271.304,E2 -22271.304} C_VEL
LIN {X 0,Y 203.543,Z 417.841,A -85,B 0,C 180,E1 -22274.118,E2 -22274.118} C_VEL
LIN {X 0,Y 199.801,Z 408.127,A -85,B 0,C 180,E1 -22277.449,E2 -22277.449} C_VEL
LIN {X 0,Y 195.46,Z 399.016,A -85,B 0,C 180,E1 -22280.625,E2 -22280.625} C_VEL
LIN {X 0,Y 191.255,Z 391.714,A -85,B 0,C 180,E1 -22283.334,E2 -22283.334} C_VEL
LIN {X 0,Y 189.238,Z 388.777,A -85,B 0,C 180,E1 -22284.529,E2 -22284.529} C_VEL
LIN {X 0,Y 188.468,Z 387.273,A -85,B 0,C 180,E1 -22285.049,E2 -22285.049} C_VEL
LIN {X 0,Y 186.407,Z 385.004,A -85,B 0,C 180,E1 -22286.184,E2 -22286.184} C_VEL
LIN {X 0,Y 185.566,Z 382.348,A -85,B 0,C 180,E1 -22286.973,E2 -22286.973} C_VEL
LIN {X 0,Y 185.578,Z 382.317,A -85,B 0,C 180,E1 -22290.575,E2 -22290.575} C_VEL
LIN {X 0,Y 185.585,Z 382.359,A -85,B 0,C 180,E1 -22295.381,E2 -22295.381} C_VEL
LIN {X 0,Y 185.672,Z 382.344,A -85,B 0,C 180,E1 -22301.132,E2 -22301.132} C_VEL
LIN {X 0,Y 185.722,Z 382.351,A -85,B 0,C 180,E1 -22304.639,E2 -22304.639} C_VEL
LIN {X 0,Y 185.939,Z 382.32,A -85,B 0,C 180,E1 -22309.327,E2 -22309.327} C_VEL
LIN {X 0,Y 185.966,Z 382.303,A -85,B 0,C 180,E1 -22313.49,E2 -22313.49} C_VEL
LIN {X 0,Y 186.207,Z 382.288,A -85,B 0,C 180,E1 -22317.836,E2 -22317.836} C_VEL
LIN {X 0,Y 186.407,Z 382.248,A -85,B 0,C 180,E1 -22320,E2 -22320} C_VEL
LIN {X 0,Y 185.926,Z 382.313,A -85,B 0,C 180,E1 -22324.335,E2 -22324.335} C_VEL
LIN {X 0,Y 186.025,Z 382.304,A -85,B 0,C 180,E1 -22328.691,E2 -22328.691} C_VEL
LIN {X 0,Y 185.761,Z 382.337,A -85,B 0,C 180,E1 -22333.12,E2 -22333.12} C_VEL
LIN {X 0,Y 185.746,Z 382.487,A -85,B 0,C 180,E1 -22338.623,E2 -22338.623} C_VEL
LIN {X 0,Y 186.469,Z 386.386,A -85,B 0,C 180,E1 -22344.493,E2 -22344.493} C_VEL
LIN {X 0,Y 187.386,Z 390.985,A -85,B 0,C 180,E1 -22350.39,E2 -22350.39} C_VEL
LIN {X 0,Y 188.225,Z 394.811,A -85,B 0,C 180,E1 -22354.773,E2 -22354.773} C_VEL
LIN {X 0,Y 189.025,Z 399.106,A -85,B 0,C 180,E1 -22359.202,E2 -22359.202} C_VEL
LIN {X 0,Y 189.549,Z 401.935,A -85,B 0,C 180,E1 -22361.96,E2 -22361.96} C_VEL
LIN {X 0,Y 190.921,Z 405.595,A -85,B 0,C 180,E1 -22362.735,E2 -22362.735} C_VEL
LIN {X 0,Y 193.051,Z 408.965,A -85,B 0,C 180,E1 -22363.764,E2 -22363.764} C_VEL
LIN {X 0,Y 194.963,Z 413.222,A -85,B 0,C 180,E1 -22364.787,E2 -22364.787} C_VEL
LIN {X 0,Y 196.018,Z 415.437,A -85,B 0,C 180,E1 -22365.345,E2 -22365.345} C_VEL
LIN {X 0,Y 198.352,Z 421.086,A -85,B 0,C 180,E1 -22366.674,E2 -22366.674} C_VEL
LIN {X 0,Y 199.28,Z 424.939,A -85,B 0,C 180,E1 -22367.408,E2 -22367.408} C_VEL
LIN {X 0,Y 200.801,Z 437.238,A -85,B 0,C 180,E1 -22369.61,E2 -22369.61} C_VEL
LIN {X 0,Y 201.293,Z 449.031,A -85,B 0,C 180,E1 -22371.871,E2 -22371.871} C_VEL
LIN {X 0,Y 200.884,Z 460.819,A -85,B 0,C 180,E1 -22374.379,E2 -22374.379} C_VEL
LIN {X 0,Y 199.615,Z 471.79,A -85,B 0,C 180,E1 -22377.048,E2 -22377.048} C_VEL
LIN {X 0,Y 197.88,Z 480.796,A -85,B 0,C 180,E1 -22379.597,E2 -22379.597} C_VEL
LIN {X 0,Y 196.042,Z 487.163,A -85,B 0,C 180,E1 -22381.642,E2 -22381.642} C_VEL
LIN {X 0,Y 192.521,Z 495.076,A -85,B 0,C 180,E1 -22384.602,E2 -22384.602} C_VEL
LIN {X 0,Y 189.051,Z 502.407,A -85,B 0,C 180,E1 -22388.178,E2 -22388.178} C_VEL
LIN {X 0,Y 186.806,Z 507.372,A -85,B 0,C 180,E1 -22391.352,E2 -22391.352} C_VEL
LIN {X 0,Y 185.181,Z 511.248,A -85,B 0,C 180,E1 -22394.595,E2 -22394.595} C_VEL
LIN {X 0,Y 184.478,Z 513.299,A -85,B 0,C 180,E1 -22396.788,E2 -22396.788} C_VEL
LIN {X 0,Y 184.081,Z 514.924,A -85,B 0,C 180,E1 -22398.997,E2 -22398.997} C_VEL
LIN {X 0,Y 184.131,Z 516.949,A -85,B 0,C 180,E1 -22403.426,E2 -22403.426} C_VEL
LIN {X 0,Y 184.442,Z 517.381,A -85,B 0,C 180,E1 -22405.631,E2 -22405.631} C_VEL
LIN {X 0,Y 184.81,Z 517.399,A -85,B 0,C 180,E1 -22407.822,E2 -22407.822} C_VEL
LIN {X 0,Y 184.997,Z 516.935,A -85,B 0,C 180,E1 -22410.002,E2 -22410.002} C_VEL
LIN {X 0,Y 184.895,Z 516.302,A -85,B 0,C 180,E1 -22411.491,E2 -22411.491} C_VEL
LIN {X 0,Y 184.517,Z 515.701,A -85,B 0,C 180,E1 -22412.689,E2 -22412.689} C_VEL
LIN {X 0,Y 183.602,Z 514.886,A -85,B 0,C 180,E1 -22413.855,E2 -22413.855} C_VEL
LIN {X 0,Y 180.93,Z 512.866,A -85,B 0,C 180,E1 -22416.124,E2 -22416.124} C_VEL
LIN {X 0,Y 178.283,Z 510.342,A -85,B 0,C 180,E1 -22418.417,E2 -22418.417} C_VEL
LIN {X 0,Y 177.213,Z 508.191,A -85,B 0,C 180,E1 -22420.188,E2 -22420.188} C_VEL
LIN {X 0,Y 177.161,Z 507.413,A -85,B 0,C 180,E1 -22420.785,E2 -22420.785} C_VEL
LIN {X 0,Y 177.955,Z 501.339,A -85,B 0,C 180,E1 -22424.876,E2 -22424.876} C_VEL
LIN {X 0,Y 179.199,Z 494.757,A -85,B 0,C 180,E1 -22428.287,E2 -22428.287} C_VEL
LIN {X 0,Y 181.428,Z 486.562,A -85,B 0,C 180,E1 -22431.614,E2 -22431.614} C_VEL
LIN {X 0,Y 182.822,Z 480.057,A -85,B 0,C 180,E1 -22433.808,E2 -22433.808} C_VEL
LIN {X 0,Y 183.862,Z 469.959,A -85,B 0,C 180,E1 -22436.69,E2 -22436.69} C_VEL
LIN {X 0,Y 184.905,Z 458.759,A -85,B 0,C 180,E1 -22439.291,E2 -22439.291} C_VEL
LIN {X 0,Y 185.338,Z 447.642,A -85,B 0,C 180,E1 -22441.428,E2 -22441.428} C_VEL
LIN {X 0,Y 185.128,Z 435.472,A -85,B 0,C 180,E1 -22443.366,E2 -22443.366} C_VEL
LIN {X 0,Y 183.959,Z 422.595,A -85,B 0,C 180,E1 -22445.1,E2 -22445.1} C_VEL
LIN {X 0,Y 181.722,Z 409.037,A -85,B 0,C 180,E1 -22446.645,E2 -22446.645} C_VEL
LIN {X 0,Y 181.054,Z 405.534,A -85,B 0,C 180,E1 -22447.036,E2 -22447.036} C_VEL
LIN {X 0,Y 181.899,Z 402.486,A -85,B 0,C 180,E1 -22449.4,E2 -22449.4} C_VEL
LIN {X 0,Y 181.496,Z 398.6,A -85,B 0,C 180,E1 -22452.631,E2 -22452.631} C_VEL
LIN {X 0,Y 180.366,Z 392.79,A -85,B 0,C 180,E1 -22457.763,E2 -22457.763} C_VEL
LIN {X 0,Y 179.368,Z 387.6,A -85,B 0,C 180,E1 -22462.724,E2 -22462.724} C_VEL
LIN {X 0,Y 178.507,Z 383.252,A -85,B 0,C 180,E1 -22467.392,E2 -22467.392} C_VEL
LIN {X 0,Y 178.49,Z 383.252,A -85,B 0,C 180,E1 -22471.804,E2 -22471.804} C_VEL
LIN {X 0,Y 178.519,Z 383.253,A -85,B 0,C 180,E1 -22476.816,E2 -22476.816} C_VEL
LIN {X 0,Y 178.676,Z 383.232,A -85,B 0,C 180,E1 -22481.66,E2 -22481.66} C_VEL
LIN {X 0,Y 178.694,Z 383.23,A -85,B 0,C 180,E1 -22486.351,E2 -22486.351} C_VEL
LIN {X 0,Y 178.984,Z 383.19,A -85,B 0,C 180,E1 -22490.964,E2 -22490.964} C_VEL
LIN {X 0,Y 179.16,Z 383.155,A -85,B 0,C 180,E1 -22497.752,E2 -22497.752} C_VEL
LIN {X 0,Y 179.377,Z 383.131,A -85,B 0,C 180,E1 -22500.001,E2 -22500.001} C_VEL
LIN {X 0,Y 178.88,Z 383.197,A -85,B 0,C 180,E1 -22504.507,E2 -22504.507} C_VEL
LIN {X 0,Y 178.981,Z 383.185,A -85,B 0,C 180,E1 -22509.037,E2 -22509.037} C_VEL
LIN {X 0,Y 178.688,Z 383.217,A -85,B 0,C 180,E1 -22513.65,E2 -22513.65} C_VEL
LIN {X 0,Y 178.63,Z 383.233,A -85,B 0,C 180,E1 -22519.216,E2 -22519.216} C_VEL
LIN {X 0,Y 178.541,Z 383.241,A -85,B 0,C 180,E1 -22525.124,E2 -22525.124} C_VEL
LIN {X 0,Y 178.529,Z 383.235,A -85,B 0,C 180,E1 -22529.994,E2 -22529.994} C_VEL
LIN {X 0,Y 178.502,Z 383.249,A -85,B 0,C 180,E1 -22534.225,E2 -22534.225} C_VEL
LIN {X 0,Y 178.425,Z 383.256,A -85,B 0,C 180,E1 -22539.068,E2 -22539.068} C_VEL
LIN {X 0,Y 178.418,Z 383.257,A -85,B 0,C 180,E1 -22542.04,E2 -22542.04} C_VEL
LIN {X 0,Y 178.406,Z 383.258,A -85,B 0,C 180,E1 -22545.161,E2 -22545.161} C_VEL
LIN {X 0,Y 178.41,Z 383.258,A -85,B 0,C 180,E1 -22548.458,E2 -22548.458} C_VEL
LIN {X 0,Y 178.428,Z 383.257,A -85,B 0,C 180,E1 -22553.782,E2 -22553.782} C_VEL
LIN {X 0,Y 178.493,Z 383.25,A -85,B 0,C 180,E1 -22556.546,E2 -22556.546} C_VEL
LIN {X 0,Y 178.518,Z 383.249,A -85,B 0,C 180,E1 -22561.751,E2 -22561.751} C_VEL
LIN {X 0,Y 179.475,Z 386.052,A -85,B 0,C 180,E1 -22562.282,E2 -22562.282} C_VEL
LIN {X 0,Y 184.095,Z 395.564,A -85,B 0,C 180,E1 -22564.484,E2 -22564.484} C_VEL
LIN {X 0,Y 187.567,Z 404.721,A -85,B 0,C 180,E1 -22566.634,E2 -22566.634} C_VEL
LIN {X 0,Y 190.71,Z 415.094,A -85,B 0,C 180,E1 -22569.242,E2 -22569.242} C_VEL
LIN {X 0,Y 191.628,Z 419.416,A -85,B 0,C 180,E1 -22570.381,E2 -22570.381} C_VEL
LIN {X 0,Y 189.362,Z 429.701,A -85,B 0,C 180,E1 -22572.726,E2 -22572.726} C_VEL
LIN {X 0,Y 187.082,Z 438.71,A -85,B 0,C 180,E1 -22575.309,E2 -22575.309} C_VEL
LIN {X 0,Y 184.591,Z 447.51,A -85,B 0,C 180,E1 -22578.468,E2 -22578.468} C_VEL
LIN {X 0,Y 182.512,Z 454.605,A -85,B 0,C 180,E1 -22581.696,E2 -22581.696} C_VEL
LIN {X 0,Y 181.17,Z 459.387,A -85,B 0,C 180,E1 -22584.433,E2 -22584.433} C_VEL
LIN {X 0,Y 179.865,Z 464.058,A -85,B 0,C 180,E1 -22587.759,E2 -22587.759} C_VEL
LIN {X 0,Y 178.85,Z 467.667,A -85,B 0,C 180,E1 -22591.124,E2 -22591.124} C_VEL
LIN {X 0,Y 178.46,Z 470.256,A -85,B 0,C 180,E1 -22594.516,E2 -22594.516} C_VEL
LIN {X 0,Y 178.473,Z 471.483,A -85,B 0,C 180,E1 -22596.783,E2 -22596.783} C_VEL
LIN {X 0,Y 178.756,Z 472.647,A -85,B 0,C 180,E1 -22600.605,E2 -22600.605} C_VEL
LIN {X 0,Y 179.266,Z 472.77,A -85,B 0,C 180,E1 -22603.603,E2 -22603.603} C_VEL
LIN {X 0,Y 179.944,Z 472.433,A -85,B 0,C 180,E1 -22605.865,E2 -22605.865} C_VEL
LIN {X 0,Y 180.779,Z 471.674,A -85,B 0,C 180,E1 -22608.118,E2 -22608.118} C_VEL
LIN {X 0,Y 181.849,Z 470.501,A -85,B 0,C 180,E1 -22610.353,E2 -22610.353} C_VEL
LIN {X 0,Y 183.701,Z 468.256,A -85,B 0,C 180,E1 -22613.335,E2 -22613.335} C_VEL
LIN {X 0,Y 186.376,Z 464.394,A -85,B 0,C 180,E1 -22616.903,E2 -22616.903} C_VEL
LIN {X 0,Y 189.266,Z 459.696,A -85,B 0,C 180,E1 -22620.084,E2 -22620.084} C_VEL
LIN {X 0,Y 192.683,Z 453.702,A -85,B 0,C 180,E1 -22623.168,E2 -22623.168} C_VEL
LIN {X 0,Y 196.551,Z 446.185,A -85,B 0,C 180,E1 -22626.154,E2 -22626.154} C_VEL
LIN {X 0,Y 200.039,Z 438.424,A -85,B 0,C 180,E1 -22628.579,E2 -22628.579} C_VEL
LIN {X 0,Y 200.756,Z 436.649,A -85,B 0,C 180,E1 -22629.058,E2 -22629.058} C_VEL
LIN {X 0,Y 200.561,Z 433.199,A -85,B 0,C 180,E1 -22630.345,E2 -22630.345} C_VEL
LIN {X 0,Y 198.776,Z 424.781,A -85,B 0,C 180,E1 -22633.528,E2 -22633.528} C_VEL
LIN {X 0,Y 196.29,Z 416.978,A -85,B 0,C 180,E1 -22636.429,E2 -22636.429} C_VEL
LIN {X 0,Y 192.746,Z 408.027,A -85,B 0,C 180,E1 -22639.735,E2 -22639.735} C_VEL
LIN {X 0,Y 189.536,Z 401.429,A -85,B 0,C 180,E1 -22642.278,E2 -22642.278} C_VEL
LIN {X 0,Y 186.676,Z 396.566,A -85,B 0,C 180,E1 -22644.299,E2 -22644.299} C_VEL
LIN {X 0,Y 184.239,Z 392.552,A -85,B 0,C 180,E1 -22646.003,E2 -22646.003} C_VEL
LIN {X 0,Y 182.383,Z 389.786,A -85,B 0,C 180,E1 -22647.243,E2 -22647.243} C_VEL
LIN {X 0,Y 181.597,Z 388.218,A -85,B 0,C 180,E1 -22647.849,E2 -22647.849} C_VEL
LIN {X 0,Y 179.469,Z 386.054,A -85,B 0,C 180,E1 -22649.152,E2 -22649.152} C_VEL
LIN {X 0,Y 178.554,Z 383.601,A -85,B 0,C 180,E1 -22649.949,E2 -22649.949} C_VEL
LIN {X 0,Y 178.499,Z 383.196,A -85,B 0,C 180,E1 -22650.109,E2 -22650.109} C_VEL
LIN {X 0,Y 178.532,Z 383.243,A -85,B 0,C 180,E1 -22654.874,E2 -22654.874} C_VEL
LIN {X 0,Y 178.62,Z 383.225,A -85,B 0,C 180,E1 -22660.783,E2 -22660.783} C_VEL
LIN {X 0,Y 178.663,Z 383.223,A -85,B 0,C 180,E1 -22664.016,E2 -22664.016} C_VEL
LIN {X 0,Y 178.891,Z 383.198,A -85,B 0,C 180,E1 -22669.152,E2 -22669.152} C_VEL
LIN {X 0,Y 178.931,Z 383.181,A -85,B 0,C 180,E1 -22673.232,E2 -22673.232} C_VEL
LIN {X 0,Y 179.153,Z 383.167,A -85,B 0,C 180,E1 -22677.751,E2 -22677.751} C_VEL
LIN {X 0,Y 179.37,Z 383.125,A -85,B 0,C 180,E1 -22679.999,E2 -22679.999} C_VEL
LIN {X 0,Y 178.874,Z 383.19,A -85,B 0,C 180,E1 -22684.506,E2 -22684.506} C_VEL
LIN {X 0,Y 178.974,Z 383.18,A -85,B 0,C 180,E1 -22689.037,E2 -22689.037} C_VEL
LIN {X 0,Y 178.684,Z 383.216,A -85,B 0,C 180,E1 -22693.65,E2 -22693.65} C_VEL
LIN {X 0,Y 178.657,Z 383.348,A -85,B 0,C 180,E1 -22696.277,E2 -22696.277} C_VEL
LIN {X 0,Y 179.023,Z 385.24,A -85,B 0,C 180,E1 -22699.584,E2 -22699.584} C_VEL
LIN {X 0,Y 179.789,Z 389.16,A -85,B 0,C 180,E1 -22705.467,E2 -22705.467} C_VEL
LIN {X 0,Y 180.683,Z 393.524,A -85,B 0,C 180,E1 -22711.163,E2 -22711.163} C_VEL
LIN {X 0,Y 181.488,Z 397.355,A -85,B 0,C 180,E1 -22715.592,E2 -22715.592} C_VEL
LIN {X 0,Y 182.081,Z 400.482,A -85,B 0,C 180,E1 -22718.891,E2 -22718.891} C_VEL
LIN {X 0,Y 183.417,Z 403.943,A -85,B 0,C 180,E1 -22719.731,E2 -22719.731} C_VEL
LIN {X 0,Y 185.759,Z 407.498,A -85,B 0,C 180,E1 -22721.008,E2 -22721.008} C_VEL
LIN {X 0,Y 187.677,Z 411.862,A -85,B 0,C 180,E1 -22722.174,E2 -22722.174} C_VEL
LIN {X 0,Y 188.899,Z 414.043,A -85,B 0,C 180,E1 -22722.854,E2 -22722.854} C_VEL
LIN {X 0,Y 191.062,Z 418.779,A -85,B 0,C 180,E1 -22724.154,E2 -22724.154} C_VEL
LIN {X 0,Y 193.54,Z 425.426,A -85,B 0,C 180,E1 -22725.822,E2 -22725.822} C_VEL
LIN {X 0,Y 194.847,Z 435.446,A -85,B 0,C 180,E1 -22727.761,E2 -22727.761} C_VEL
LIN {X 0,Y 195.359,Z 447.502,A -85,B 0,C 180,E1 -22730.189,E2 -22730.189} C_VEL
LIN {X 0,Y 194.976,Z 457.91,A -85,B 0,C 180,E1 -22732.467,E2 -22732.467} C_VEL
LIN {X 0,Y 193.961,Z 467.777,A -85,B 0,C 180,E1 -22734.887,E2 -22734.887} C_VEL
LIN {X 0,Y 192.108,Z 478.009,A -85,B 0,C 180,E1 -22737.763,E2 -22737.763} C_VEL
LIN {X 0,Y 189.721,Z 486.64,A -85,B 0,C 180,E1 -22740.607,E2 -22740.607} C_VEL
LIN {X 0,Y 186.678,Z 493.282,A -85,B 0,C 180,E1 -22743.144,E2 -22743.144} C_VEL
LIN {X 0,Y 183.402,Z 499.869,A -85,B 0,C 180,E1 -22746.276,E2 -22746.276} C_VEL
LIN {X 0,Y 180.747,Z 505.165,A -85,B 0,C 180,E1 -22749.518,E2 -22749.518} C_VEL
LIN {X 0,Y 178.813,Z 509.353,A -85,B 0,C 180,E1 -22752.858,E2 -22752.858} C_VEL
LIN {X 0,Y 177.522,Z 512.523,A -85,B 0,C 180,E1 -22756.261,E2 -22756.261} C_VEL
LIN {X 0,Y 176.903,Z 515.289,A -85,B 0,C 180,E1 -22760.858,E2 -22760.858} C_VEL
LIN {X 0,Y 177.067,Z 516.098,A -85,B 0,C 180,E1 -22763.163,E2 -22763.163} C_VEL
LIN {X 0,Y 177.355,Z 516.511,A -85,B 0,C 180,E1 -22765.456,E2 -22765.456} C_VEL
LIN {X 0,Y 177.75,Z 516.497,A -85,B 0,C 180,E1 -22767.736,E2 -22767.736} C_VEL
LIN {X 0,Y 177.948,Z 516.013,A -85,B 0,C 180,E1 -22770.002,E2 -22770.002} C_VEL
LIN {X 0,Y 177.831,Z 515.066,A -85,B 0,C 180,E1 -22772.267,E2 -22772.267} C_VEL
LIN {X 0,Y 177.461,Z 513.655,A -85,B 0,C 180,E1 -22774.545,E2 -22774.545} C_VEL
LIN {X 0,Y 177.156,Z 511.264,A -85,B 0,C 180,E1 -22777.352,E2 -22777.352} C_VEL
LIN {X 0,Y 177.161,Z 507.413,A -85,B 0,C 180,E1 -22780.785,E2 -22780.785} C_VEL
LIN {X 0,Y 176.688,Z 505.01,A -85,B 0,C 180,E1 -22782.528,E2 -22782.528} C_VEL
LIN {X 0,Y 174.433,Z 500.528,A -85,B 0,C 180,E1 -22785.329,E2 -22785.329} C_VEL
LIN {X 0,Y 172.609,Z 495.475,A -85,B 0,C 180,E1 -22788.085,E2 -22788.085} C_VEL
LIN {X 0,Y 172.815,Z 492.109,A -85,B 0,C 180,E1 -22789.701,E2 -22789.701} C_VEL
LIN {X 0,Y 175.221,Z 483.727,A -85,B 0,C 180,E1 -22793.065,E2 -22793.065} C_VEL
LIN {X 0,Y 176.234,Z 476.793,A -85,B 0,C 180,E1 -22795.387,E2 -22795.387} C_VEL
LIN {X 0,Y 177.514,Z 466.197,A -85,B 0,C 180,E1 -22798.367,E2 -22798.367} C_VEL
LIN {X 0,Y 178.454,Z 455.585,A -85,B 0,C 180,E1 -22800.797,E2 -22800.797} C_VEL
LIN {X 0,Y 178.835,Z 443.835,A -85,B 0,C 180,E1 -22803.045,E2 -22803.045} C_VEL
LIN {X 0,Y 178.381,Z 430.905,A -85,B 0,C 180,E1 -22805.123,E2 -22805.123} C_VEL
LIN {X 0,Y 176.814,Z 417.549,A -85,B 0,C 180,E1 -22806.934,E2 -22806.934} C_VEL
LIN {X 0,Y 174.456,Z 404.716,A -85,B 0,C 180,E1 -22808.409,E2 -22808.409} C_VEL
LIN {X 0,Y 174.857,Z 402.518,A -85,B 0,C 180,E1 -22810.212,E2 -22810.212} C_VEL
LIN {X 0,Y 173.991,Z 397.087,A -85,B 0,C 180,E1 -22815.019,E2 -22815.019} C_VEL
LIN {X 0,Y 173.041,Z 392.404,A -85,B 0,C 180,E1 -22819.471,E2 -22819.471} C_VEL
LIN {X 0,Y 172.258,Z 388.186,A -85,B 0,C 180,E1 -22823.732,E2 -22823.732} C_VEL
LIN {X 0,Y 171.462,Z 384.126,A -85,B 0,C 180,E1 -22828.262,E2 -22828.262} C_VEL
LIN {X 0,Y 171.423,Z 384.134,A -85,B 0,C 180,E1 -22833.194,E2 -22833.194} C_VEL
LIN {X 0,Y 171.472,Z 384.13,A -85,B 0,C 180,E1 -22838.354,E2 -22838.354} C_VEL
LIN {X 0,Y 171.601,Z 384.115,A -85,B 0,C 180,E1 -22840.875,E2 -22840.875} C_VEL
LIN {X 0,Y 171.619,Z 384.11,A -85,B 0,C 180,E1 -22845.777,E2 -22845.777} C_VEL
LIN {X 0,Y 171.916,Z 384.071,A -85,B 0,C 180,E1 -22850.589,E2 -22850.589} C_VEL
LIN {X 0,Y 171.831,Z 384.079,A -85,B 0,C 180,E1 -22855.308,E2 -22855.308} C_VEL
LIN {X 0,Y 172.339,Z 384.007,A -85,B 0,C 180,E1 -22860.001,E2 -22860.001} C_VEL
LIN {X 0,Y 171.83,Z 384.075,A -85,B 0,C 180,E1 -22864.693,E2 -22864.693} C_VEL
LIN {X 0,Y 171.914,Z 384.065,A -85,B 0,C 180,E1 -22869.412,E2 -22869.412} C_VEL
LIN {X 0,Y 171.601,Z 384.096,A -85,B 0,C 180,E1 -22874.226,E2 -22874.226} C_VEL
LIN {X 0,Y 171.551,Z 384.116,A -85,B 0,C 180,E1 -22879.562,E2 -22879.562} C_VEL
LIN {X 0,Y 171.476,Z 384.123,A -85,B 0,C 180,E1 -22885.616,E2 -22885.616} C_VEL
LIN {X 0,Y 171.448,Z 384.117,A -85,B 0,C 180,E1 -22890.587,E2 -22890.587} C_VEL
LIN {X 0,Y 171.413,Z 384.132,A -85,B 0,C 180,E1 -22895.031,E2 -22895.031} C_VEL
LIN {X 0,Y 171.386,Z 384.132,A -85,B 0,C 180,E1 -22898.816,E2 -22898.816} C_VEL
LIN {X 0,Y 171.336,Z 384.138,A -85,B 0,C 180,E1 -22904.214,E2 -22904.214} C_VEL
LIN {X 0,Y 171.342,Z 384.14,A -85,B 0,C 180,E1 -22908.981,E2 -22908.981} C_VEL
LIN {X 0,Y 171.393,Z 384.132,A -85,B 0,C 180,E1 -22912.04,E2 -22912.04} C_VEL
LIN {X 0,Y 171.404,Z 384.132,A -85,B 0,C 180,E1 -22915.091,E2 -22915.091} C_VEL
LIN {X 0,Y 171.502,Z 384.194,A -85,B 0,C 180,E1 -22920.231,E2 -22920.231} C_VEL
LIN {X 0,Y 172.56,Z 387.097,A -85,B 0,C 180,E1 -22920.831,E2 -22920.831} C_VEL
LIN {X 0,Y 175.902,Z 393.792,A -85,B 0,C 180,E1 -22922.481,E2 -22922.481} C_VEL
LIN {X 0,Y 179.669,Z 402.593,A -85,B 0,C 180,E1 -22924.7,E2 -22924.7} C_VEL
LIN {X 0,Y 183.096,Z 413.082,A -85,B 0,C 180,E1 -22927.426,E2 -22927.426} C_VEL
LIN {X 0,Y 185.074,Z 421.066,A -85,B 0,C 180,E1 -22929.654,E2 -22929.654} C_VEL
LIN {X 0,Y 182.697,Z 431.171,A -85,B 0,C 180,E1 -22932.075,E2 -22932.075} C_VEL
LIN {X 0,Y 180.31,Z 440.08,A -85,B 0,C 180,E1 -22934.744,E2 -22934.744} C_VEL
LIN {X 0,Y 177.711,Z 448.798,A -85,B 0,C 180,E1 -22938.015,E2 -22938.015} C_VEL
LIN {X 0,Y 175.556,Z 455.803,A -85,B 0,C 180,E1 -22941.364,E2 -22941.364} C_VEL
LIN {X 0,Y 173.628,Z 462.191,A -85,B 0,C 180,E1 -22945.355,E2 -22945.355} C_VEL
LIN {X 0,Y 172.421,Z 466.434,A -85,B 0,C 180,E1 -22948.831,E2 -22948.831} C_VEL
LIN {X 0,Y 171.561,Z 469.652,A -85,B 0,C 180,E1 -22952.346,E2 -22952.346} C_VEL
LIN {X 0,Y 171.412,Z 471.242,A -85,B 0,C 180,E1 -22954.702,E2 -22954.702} C_VEL
LIN {X 0,Y 171.433,Z 472.44,A -85,B 0,C 180,E1 -22957.063,E2 -22957.063} C_VEL
LIN {X 0,Y 171.855,Z 473.614,A -85,B 0,C 180,E1 -22961.797,E2 -22961.797} C_VEL
LIN {X 0,Y 173.094,Z 473.267,A -85,B 0,C 180,E1 -22966.51,E2 -22966.51} C_VEL
LIN {X 0,Y 175.181,Z 471.267,A -85,B 0,C 180,E1 -22971.164,E2 -22971.164} C_VEL
LIN {X 0,Y 177.003,Z 469.163,A -85,B 0,C 180,E1 -22974.042,E2 -22974.042} C_VEL
LIN {X 0,Y 180.017,Z 465.053,A -85,B 0,C 180,E1 -22977.934,E2 -22977.934} C_VEL
LIN {X 0,Y 183.102,Z 460.295,A -85,B 0,C 180,E1 -22981.208,E2 -22981.208} C_VEL
LIN {X 0,Y 186.739,Z 454.233,A -85,B 0,C 180,E1 -22984.368,E2 -22984.368} C_VEL
LIN {X 0,Y 190.803,Z 446.612,A -85,B 0,C 180,E1 -22987.426,E2 -22987.426} C_VEL
LIN {X 0,Y 194.468,Z 438.754,A -85,B 0,C 180,E1 -22989.897,E2 -22989.897} C_VEL
LIN {X 0,Y 194.233,Z 434.915,A -85,B 0,C 180,E1 -22991.439,E2 -22991.439} C_VEL
LIN {X 0,Y 192.615,Z 426.968,A -85,B 0,C 180,E1 -22994.656,E2 -22994.656} C_VEL
LIN {X 0,Y 189.851,Z 418.036,A -85,B 0,C 180,E1 -22998.214,E2 -22998.214} C_VEL
LIN {X 0,Y 186.558,Z 409.661,A -85,B 0,C 180,E1 -23001.567,E2 -23001.567} C_VEL
LIN {X 0,Y 182.768,Z 402.292,A -85,B 0,C 180,E1 -23004.774,E2 -23004.774} C_VEL
LIN {X 0,Y 180.098,Z 397.73,A -85,B 0,C 180,E1 -23006.884,E2 -23006.884} C_VEL
LIN {X 0,Y 178.137,Z 394.196,A -85,B 0,C 180,E1 -23008.482,E2 -23008.482} C_VEL
LIN {X 0,Y 175.963,Z 391.597,A -85,B 0,C 180,E1 -23010.028,E2 -23010.028} C_VEL
LIN {X 0,Y 175.018,Z 389.351,A -85,B 0,C 180,E1 -23010.927,E2 -23010.927} C_VEL
LIN {X 0,Y 172.635,Z 387.249,A -85,B 0,C 180,E1 -23012.578,E2 -23012.578} C_VEL
LIN {X 0,Y 171.587,Z 384.884,A -85,B 0,C 180,E1 -23013.577,E2 -23013.577} C_VEL
LIN {X 0,Y 171.452,Z 384.121,A -85,B 0,C 180,E1 -23013.821,E2 -23013.821} C_VEL
LIN {X 0,Y 171.459,Z 384.116,A -85,B 0,C 180,E1 -23018.351,E2 -23018.351} C_VEL
LIN {X 0,Y 171.576,Z 384.101,A -85,B 0,C 180,E1 -23020.871,E2 -23020.871} C_VEL
LIN {X 0,Y 171.607,Z 384.107,A -85,B 0,C 180,E1 -23025.775,E2 -23025.775} C_VEL
LIN {X 0,Y 171.907,Z 384.068,A -85,B 0,C 180,E1 -23030.588,E2 -23030.588} C_VEL
LIN {X 0,Y 171.824,Z 384.064,A -85,B 0,C 180,E1 -23035.307,E2 -23035.307} C_VEL
LIN {X 0,Y 172.332,Z 384.001,A -85,B 0,C 180,E1 -23039.999,E2 -23039.999} C_VEL
LIN {X 0,Y 171.823,Z 384.068,A -85,B 0,C 180,E1 -23044.692,E2 -23044.692} C_VEL
LIN {X 0,Y 171.906,Z 384.058,A -85,B 0,C 180,E1 -23049.411,E2 -23049.411} C_VEL
LIN {X 0,Y 171.67,Z 384.184,A -85,B 0,C 180,E1 -23053.615,E2 -23053.615} C_VEL
LIN {X 0,Y 172.235,Z 387.076,A -85,B 0,C 180,E1 -23059.052,E2 -23059.052} C_VEL
LIN {X 0,Y 172.738,Z 390.192,A -85,B 0,C 180,E1 -23064.007,E2 -23064.007} C_VEL
LIN {X 0,Y 173.473,Z 393.826,A -85,B 0,C 180,E1 -23069.088,E2 -23069.088} C_VEL
LIN {X 0,Y 174.448,Z 398.024,A -85,B 0,C 180,E1 -23074.334,E2 -23074.334} C_VEL
LIN {X 0,Y 174.581,Z 398.839,A -85,B 0,C 180,E1 -23075.227,E2 -23075.227} C_VEL
LIN {X 0,Y 175.974,Z 402.38,A -85,B 0,C 180,E1 -23076.254,E2 -23076.254} C_VEL
LIN {X 0,Y 178.61,Z 406.329,A -85,B 0,C 180,E1 -23077.916,E2 -23077.916} C_VEL
LIN {X 0,Y 180.671,Z 410.816,A -85,B 0,C 180,E1 -23079.331,E2 -23079.331} C_VEL
LIN {X 0,Y 181.985,Z 413.161,A -85,B 0,C 180,E1 -23080.159,E2 -23080.159} C_VEL
LIN {X 0,Y 184.161,Z 417.837,A -85,B 0,C 180,E1 -23081.625,E2 -23081.625} C_VEL
LIN {X 0,Y 188.159,Z 427.982,A -85,B 0,C 180,E1 -23084.529,E2 -23084.529} C_VEL
LIN {X 0,Y 188.797,Z 431.115,A -85,B 0,C 180,E1 -23085.263,E2 -23085.263} C_VEL
LIN {X 0,Y 189.531,Z 443.635,A -85,B 0,C 180,E1 -23087.869,E2 -23087.869} C_VEL
LIN {X 0,Y 189.224,Z 455.593,A -85,B 0,C 180,E1 -23090.574,E2 -23090.574} C_VEL
LIN {X 0,Y 188.032,Z 466.321,A -85,B 0,C 180,E1 -23093.273,E2 -23093.273} C_VEL
LIN {X 0,Y 186.138,Z 476.342,A -85,B 0,C 180,E1 -23096.165,E2 -23096.165} C_VEL
LIN {X 0,Y 183.913,Z 484.596,A -85,B 0,C 180,E1 -23098.945,E2 -23098.945} C_VEL
LIN {X 0,Y 181.661,Z 490.195,A -85,B 0,C 180,E1 -23101.082,E2 -23101.082} C_VEL
LIN {X 0,Y 177.374,Z 498.206,A -85,B 0,C 180,E1 -23104.792,E2 -23104.792} C_VEL
LIN {X 0,Y 174.038,Z 504.455,A -85,B 0,C 180,E1 -23108.69,E2 -23108.69} C_VEL
LIN {X 0,Y 171.986,Z 508.602,A -85,B 0,C 180,E1 -23112.155,E2 -23112.155} C_VEL
LIN {X 0,Y 170.565,Z 511.737,A -85,B 0,C 180,E1 -23115.688,E2 -23115.688} C_VEL
LIN {X 0,Y 169.841,Z 514.453,A -85,B 0,C 180,E1 -23120.474,E2 -23120.474} C_VEL
LIN {X 0,Y 169.983,Z 515.244,A -85,B 0,C 180,E1 -23122.877,E2 -23122.877} C_VEL
LIN {X 0,Y 170.272,Z 515.639,A -85,B 0,C 180,E1 -23125.267,E2 -23125.267} C_VEL
LIN {X 0,Y 170.688,Z 515.592,A -85,B 0,C 180,E1 -23127.642,E2 -23127.642} C_VEL
LIN {X 0,Y 170.9,Z 515.091,A -85,B 0,C 180,E1 -23130.002,E2 -23130.002} C_VEL
LIN {X 0,Y 170.748,Z 514.121,A -85,B 0,C 180,E1 -23132.361,E2 -23132.361} C_VEL
LIN {X 0,Y 170.355,Z 512.681,A -85,B 0,C 180,E1 -23134.735,E2 -23134.735} C_VEL
LIN {X 0,Y 170.038,Z 509.632,A -85,B 0,C 180,E1 -23138.318,E2 -23138.318} C_VEL
LIN {X 0,Y 170.209,Z 505.506,A -85,B 0,C 180,E1 -23141.916,E2 -23141.916} C_VEL
LIN {X 0,Y 171.224,Z 499.19,A -85,B 0,C 180,E1 -23146.086,E2 -23146.086} C_VEL
LIN {X 0,Y 172.815,Z 492.109,A -85,B 0,C 180,E1 -23149.701,E2 -23149.701} C_VEL
LIN {X 0,Y 173.122,Z 489.768,A -85,B 0,C 180,E1 -23150.749,E2 -23150.749} C_VEL
LIN {X 0,Y 172.644,Z 486.143,A -85,B 0,C 180,E1 -23152.304,E2 -23152.304} C_VEL
LIN {X 0,Y 169.981,Z 475.787,A -85,B 0,C 180,E1 -23156.294,E2 -23156.294} C_VEL
LIN {X 0,Y 170.086,Z 471.426,A -85,B 0,C 180,E1 -23157.687,E2 -23157.687} C_VEL
LIN {X 0,Y 171.416,Z 460.602,A -85,B 0,C 180,E1 -23160.572,E2 -23160.572} C_VEL
LIN {X 0,Y 172.177,Z 449.104,A -85,B 0,C 180,E1 -23163.091,E2 -23163.091} C_VEL
LIN {X 0,Y 172.264,Z 436.956,A -85,B 0,C 180,E1 -23165.318,E2 -23165.318} C_VEL
LIN {X 0,Y 171.362,Z 423.699,A -85,B 0,C 180,E1 -23167.383,E2 -23167.383} C_VEL
LIN {X 0,Y 169.176,Z 410.024,A -85,B 0,C 180,E1 -23169.225,E2 -23169.225} C_VEL
LIN {X 0,Y 167.799,Z 403.737,A -85,B 0,C 180,E1 -23170.016,E2 -23170.016} C_VEL
LIN {X 0,Y 167.121,Z 399.006,A -85,B 0,C 180,E1 -23174.365,E2 -23174.365} C_VEL
LIN {X 0,Y 166.062,Z 393.652,A -85,B 0,C 180,E1 -23179.625,E2 -23179.625} C_VEL
LIN {X 0,Y 165.314,Z 389.626,A -85,B 0,C 180,E1 -23183.88,E2 -23183.88} C_VEL
LIN {X 0,Y 164.414,Z 385.006,A -85,B 0,C 180,E1 -23189.318,E2 -23189.318} C_VEL
LIN {X 0,Y 164.421,Z 385.007,A -85,B 0,C 180,E1 -23194.695,E2 -23194.695} C_VEL
LIN {X 0,Y 164.491,Z 385,A -85,B 0,C 180,E1 -23200.051,E2 -23200.051} C_VEL
LIN {X 0,Y 164.564,Z 384.989,A -85,B 0,C 180,E1 -23205.153,E2 -23205.153} C_VEL
LIN {X 0,Y 164.859,Z 384.95,A -85,B 0,C 180,E1 -23210.182,E2 -23210.182} C_VEL
LIN {X 0,Y 164.868,Z 384.948,A -85,B 0,C 180,E1 -23212.653,E2 -23212.653} C_VEL
LIN {X 0,Y 165.056,Z 384.911,A -85,B 0,C 180,E1 -23217.56,E2 -23217.56} C_VEL
LIN {X 0,Y 165.302,Z 384.883,A -85,B 0,C 180,E1 -23220.001,E2 -23220.001} C_VEL
LIN {X 0,Y 164.78,Z 384.952,A -85,B 0,C 180,E1 -23224.894,E2 -23224.894} C_VEL
LIN {X 0,Y 164.857,Z 384.946,A -85,B 0,C 180,E1 -23229.819,E2 -23229.819} C_VEL
LIN {X 0,Y 164.543,Z 384.972,A -85,B 0,C 180,E1 -23234.85,E2 -23234.85} C_VEL
LIN {X 0,Y 164.48,Z 384.995,A -85,B 0,C 180,E1 -23239.989,E2 -23239.989} C_VEL
LIN {X 0,Y 164.4,Z 385.007,A -85,B 0,C 180,E1 -23246.134,E2 -23246.134} C_VEL
LIN {X 0,Y 164.382,Z 384.999,A -85,B 0,C 180,E1 -23251.228,E2 -23251.228} C_VEL
LIN {X 0,Y 164.319,Z 385.016,A -85,B 0,C 180,E1 -23256.784,E2 -23256.784} C_VEL
LIN {X 0,Y 164.307,Z 385.017,A -85,B 0,C 180,E1 -23259.913,E2 -23259.913} C_VEL
LIN {X 0,Y 164.285,Z 385.019,A -85,B 0,C 180,E1 -23263.341,E2 -23263.341} C_VEL
LIN {X 0,Y 164.298,Z 385.016,A -85,B 0,C 180,E1 -23266.808,E2 -23266.808} C_VEL
LIN {X 0,Y 164.301,Z 385.014,A -85,B 0,C 180,E1 -23270.351,E2 -23270.351} C_VEL
LIN {X 0,Y 164.336,Z 385.012,A -85,B 0,C 180,E1 -23274.348,E2 -23274.348} C_VEL
LIN {X 0,Y 164.39,Z 385.025,A -85,B 0,C 180,E1 -23278.5,E2 -23278.5} C_VEL
LIN {X 0,Y 165.421,Z 387.891,A -85,B 0,C 180,E1 -23279.138,E2 -23279.138} C_VEL
LIN {X 0,Y 166.357,Z 389.119,A -85,B 0,C 180,E1 -23279.536,E2 -23279.536} C_VEL
LIN {X 0,Y 171.641,Z 400.611,A -85,B 0,C 180,E1 -23282.596,E2 -23282.596} C_VEL
LIN {X 0,Y 175.126,Z 410.072,A -85,B 0,C 180,E1 -23285.186,E2 -23285.186} C_VEL
LIN {X 0,Y 177.569,Z 418.647,A -85,B 0,C 180,E1 -23287.646,E2 -23287.646} C_VEL
LIN {X 0,Y 178.488,Z 422.715,A -85,B 0,C 180,E1 -23288.87,E2 -23288.87} C_VEL
LIN {X 0,Y 176.052,Z 432.638,A -85,B 0,C 180,E1 -23291.374,E2 -23291.374} C_VEL
LIN {X 0,Y 173.554,Z 441.45,A -85,B 0,C 180,E1 -23294.135,E2 -23294.135} C_VEL
LIN {X 0,Y 170.843,Z 450.085,A -85,B 0,C 180,E1 -23297.526,E2 -23297.526} C_VEL
LIN {X 0,Y 168.589,Z 456.988,A -85,B 0,C 180,E1 -23301.004,E2 -23301.004} C_VEL
LIN {X 0,Y 166.601,Z 463.313,A -85,B 0,C 180,E1 -23305.158,E2 -23305.158} C_VEL
LIN {X 0,Y 165.349,Z 467.501,A -85,B 0,C 180,E1 -23308.78,E2 -23308.78} C_VEL
LIN {X 0,Y 164.496,Z 470.664,A -85,B 0,C 180,E1 -23312.447,E2 -23312.447} C_VEL
LIN {X 0,Y 164.367,Z 472.229,A -85,B 0,C 180,E1 -23314.904,E2 -23314.904} C_VEL
LIN {X 0,Y 164.398,Z 473.383,A -85,B 0,C 180,E1 -23317.367,E2 -23317.367} C_VEL
LIN {X 0,Y 164.91,Z 474.504,A -85,B 0,C 180,E1 -23322.301,E2 -23322.301} C_VEL
LIN {X 0,Y 165.458,Z 474.504,A -85,B 0,C 180,E1 -23324.763,E2 -23324.763} C_VEL
LIN {X 0,Y 166.259,Z 474.09,A -85,B 0,C 180,E1 -23327.21,E2 -23327.21} C_VEL
LIN {X 0,Y 168.553,Z 472.033,A -85,B 0,C 180,E1 -23332.039,E2 -23332.039} C_VEL
LIN {X 0,Y 170.33,Z 470.073,A -85,B 0,C 180,E1 -23334.802,E2 -23334.802} C_VEL
LIN {X 0,Y 173.708,Z 465.715,A -85,B 0,C 180,E1 -23339.044,E2 -23339.044} C_VEL
LIN {X 0,Y 177.023,Z 460.893,A -85,B 0,C 180,E1 -23342.407,E2 -23342.407} C_VEL
LIN {X 0,Y 180.885,Z 454.763,A -85,B 0,C 180,E1 -23345.646,E2 -23345.646} C_VEL
LIN {X 0,Y 185.161,Z 447.027,A -85,B 0,C 180,E1 -23348.774,E2 -23348.774} C_VEL
LIN {X 0,Y 188.292,Z 440.586,A -85,B 0,C 180,E1 -23350.879,E2 -23350.879} C_VEL
LIN {X 0,Y 187.492,Z 433.72,A -85,B 0,C 180,E1 -23353.886,E2 -23353.886} C_VEL
LIN {X 0,Y 185.721,Z 426.396,A -85,B 0,C 180,E1 -23357.065,E2 -23357.065} C_VEL
LIN {X 0,Y 183.658,Z 419.669,A -85,B 0,C 180,E1 -23359.934,E2 -23359.934} C_VEL
LIN {X 0,Y 181.171,Z 413.174,A -85,B 0,C 180,E1 -23362.783,E2 -23362.783} C_VEL
LIN {X 0,Y 176.902,Z 404.491,A -85,B 0,C 180,E1 -23366.888,E2 -23366.888} C_VEL
LIN {X 0,Y 174.497,Z 400.073,A -85,B 0,C 180,E1 -23369.101,E2 -23369.101} C_VEL
LIN {X 0,Y 172.503,Z 397.436,A -85,B 0,C 180,E1 -23370.731,E2 -23370.731} C_VEL
LIN {X 0,Y 171.185,Z 395.076,A -85,B 0,C 180,E1 -23371.993,E2 -23371.993} C_VEL
LIN {X 0,Y 169.161,Z 392.547,A -85,B 0,C 180,E1 -23373.708,E2 -23373.708} C_VEL
LIN {X 0,Y 168.229,Z 390.417,A -85,B 0,C 180,E1 -23374.732,E2 -23374.732} C_VEL
LIN {X 0,Y 165.719,Z 388.337,A -85,B 0,C 180,E1 -23376.82,E2 -23376.82} C_VEL
LIN {X 0,Y 164.621,Z 386.028,A -85,B 0,C 180,E1 -23378.064,E2 -23378.064} C_VEL
LIN {X 0,Y 164.416,Z 384.994,A -85,B 0,C 180,E1 -23378.448,E2 -23378.448} C_VEL
LIN {X 0,Y 164.502,Z 384.976,A -85,B 0,C 180,E1 -23382.598,E2 -23382.598} C_VEL
LIN {X 0,Y 164.776,Z 384.958,A -85,B 0,C 180,E1 -23388.801,E2 -23388.801} C_VEL
LIN {X 0,Y 164.859,Z 384.937,A -85,B 0,C 180,E1 -23392.652,E2 -23392.652} C_VEL
LIN {X 0,Y 165.049,Z 384.925,A -85,B 0,C 180,E1 -23397.559,E2 -23397.559} C_VEL
LIN {X 0,Y 165.294,Z 384.877,A -85,B 0,C 180,E1 -23399.999,E2 -23399.999} C_VEL
LIN {X 0,Y 164.773,Z 384.945,A -85,B 0,C 180,E1 -23404.893,E2 -23404.893} C_VEL
LIN {X 0,Y 164.849,Z 384.936,A -85,B 0,C 180,E1 -23409.818,E2 -23409.818} C_VEL
LIN {X 0,Y 164.815,Z 385.324,A -85,B 0,C 180,E1 -23411.267,E2 -23411.267} C_VEL
LIN {X 0,Y 165.28,Z 388.282,A -85,B 0,C 180,E1 -23417.316,E2 -23417.316} C_VEL
LIN {X 0,Y 165.725,Z 391.242,A -85,B 0,C 180,E1 -23422.437,E2 -23422.437} C_VEL
LIN {X 0,Y 166.432,Z 394.75,A -85,B 0,C 180,E1 -23427.678,E2 -23427.678} C_VEL
LIN {X 0,Y 166.93,Z 396.881,A -85,B 0,C 180,E1 -23430.608,E2 -23430.608} C_VEL
LIN {X 0,Y 168.374,Z 400.459,A -85,B 0,C 180,E1 -23431.912,E2 -23431.912} C_VEL
LIN {X 0,Y 171.437,Z 404.856,A -85,B 0,C 180,E1 -23434.221,E2 -23434.221} C_VEL
LIN {X 0,Y 173.401,Z 409.207,A -85,B 0,C 180,E1 -23435.823,E2 -23435.823} C_VEL
LIN {X 0,Y 174.977,Z 411.847,A -85,B 0,C 180,E1 -23436.952,E2 -23436.952} C_VEL
LIN {X 0,Y 177.255,Z 416.77,A -85,B 0,C 180,E1 -23438.714,E2 -23438.714} C_VEL
LIN {X 0,Y 180.621,Z 424.983,A -85,B 0,C 180,E1 -23441.412,E2 -23441.412} C_VEL
LIN {X 0,Y 183.228,Z 432.248,A -85,B 0,C 180,E1 -23443.663,E2 -23443.663} C_VEL
LIN {X 0,Y 183.749,Z 438.968,A -85,B 0,C 180,E1 -23445.197,E2 -23445.197} C_VEL
LIN {X 0,Y 183.7,Z 449.54,A -85,B 0,C 180,E1 -23447.623,E2 -23447.623} C_VEL
LIN {X 0,Y 182.878,Z 459.986,A -85,B 0,C 180,E1 -23450.228,E2 -23450.228} C_VEL
LIN {X 0,Y 181.292,Z 470.16,A -85,B 0,C 180,E1 -23453.069,E2 -23453.069} C_VEL
LIN {X 0,Y 179.096,Z 479.51,A -85,B 0,C 180,E1 -23456.077,E2 -23456.077} C_VEL
LIN {X 0,Y 176.647,Z 486.944,A -85,B 0,C 180,E1 -23458.857,E2 -23458.857} C_VEL
LIN {X 0,Y 173.4,Z 493.258,A -85,B 0,C 180,E1 -23461.562,E2 -23461.562} C_VEL
LIN {X 0,Y 170.383,Z 498.554,A -85,B 0,C 180,E1 -23464.337,E2 -23464.337} C_VEL
LIN {X 0,Y 167.393,Z 503.748,A -85,B 0,C 180,E1 -23467.8,E2 -23467.8} C_VEL
LIN {X 0,Y 165.193,Z 507.849,A -85,B 0,C 180,E1 -23471.394,E2 -23471.394} C_VEL
LIN {X 0,Y 163.639,Z 510.946,A -85,B 0,C 180,E1 -23475.069,E2 -23475.069} C_VEL
LIN {X 0,Y 162.813,Z 513.619,A -85,B 0,C 180,E1 -23480.059,E2 -23480.059} C_VEL
LIN {X 0,Y 162.922,Z 514.455,A -85,B 0,C 180,E1 -23482.817,E2 -23482.817} C_VEL
LIN {X 0,Y 163.625,Z 514.688,A -85,B 0,C 180,E1 -23487.54,E2 -23487.54} C_VEL
LIN {X 0,Y 163.852,Z 514.17,A -85,B 0,C 180,E1 -23490.002,E2 -23490.002} C_VEL
LIN {X 0,Y 163.65,Z 513.172,A -85,B 0,C 180,E1 -23492.463,E2 -23492.463} C_VEL
LIN {X 0,Y 163.248,Z 511.699,A -85,B 0,C 180,E1 -23494.941,E2 -23494.941} C_VEL
LIN {X 0,Y 162.981,Z 508.612,A -85,B 0,C 180,E1 -23498.682,E2 -23498.682} C_VEL
LIN {X 0,Y 163.228,Z 504.441,A -85,B 0,C 180,E1 -23502.434,E2 -23502.434} C_VEL
LIN {X 0,Y 164.333,Z 498.048,A -85,B 0,C 180,E1 -23506.781,E2 -23506.781} C_VEL
LIN {X 0,Y 166.046,Z 491.111,A -85,B 0,C 180,E1 -23510.439,E2 -23510.439} C_VEL
LIN {X 0,Y 168.537,Z 482.707,A -85,B 0,C 180,E1 -23513.926,E2 -23513.926} C_VEL
LIN {X 0,Y 169.799,Z 473.427,A -85,B 0,C 180,E1 -23517.086,E2 -23517.086} C_VEL
LIN {X 0,Y 170.086,Z 471.426,A -85,B 0,C 180,E1 -23517.687,E2 -23517.687} C_VEL
LIN {X 0,Y 170.139,Z 467.042,A -85,B 0,C 180,E1 -23519.016,E2 -23519.016} C_VEL
LIN {X 0,Y 168.295,Z 459.84,A -85,B 0,C 180,E1 -23521.239,E2 -23521.239} C_VEL
LIN {X 0,Y 166.17,Z 452.309,A -85,B 0,C 180,E1 -23523.375,E2 -23523.375} C_VEL
LIN {X 0,Y 165.775,Z 447.367,A -85,B 0,C 180,E1 -23524.528,E2 -23524.528} C_VEL
LIN {X 0,Y 165.864,Z 435.923,A -85,B 0,C 180,E1 -23526.711,E2 -23526.711} C_VEL
LIN {X 0,Y 165.09,Z 424.323,A -85,B 0,C 180,E1 -23528.64,E2 -23528.64} C_VEL
LIN {X 0,Y 163.345,Z 412.175,A -85,B 0,C 180,E1 -23530.437,E2 -23530.437} C_VEL
LIN {X 0,Y 162.047,Z 406.904,A -85,B 0,C 180,E1 -23531.218,E2 -23531.218} C_VEL
LIN {X 0,Y 160.726,Z 403.643,A -85,B 0,C 180,E1 -23531.802,E2 -23531.802} C_VEL
LIN {X 0,Y 160.54,Z 402.606,A -85,B 0,C 180,E1 -23531.96,E2 -23531.96} C_VEL
LIN {X 0,Y 159.928,Z 399.189,A -85,B 0,C 180,E1 -23535.323,E2 -23535.323} C_VEL
LIN {X 0,Y 159.033,Z 394.552,A -85,B 0,C 180,E1 -23540.159,E2 -23540.159} C_VEL
LIN {X 0,Y 158.25,Z 390.474,A -85,B 0,C 180,E1 -23544.737,E2 -23544.737} C_VEL
LIN {X 0,Y 157.374,Z 385.882,A -85,B 0,C 180,E1 -23550.395,E2 -23550.395} C_VEL
LIN {X 0,Y 157.32,Z 385.893,A -85,B 0,C 180,E1 -23556.293,E2 -23556.293} C_VEL
LIN {X 0,Y 157.438,Z 385.879,A -85,B 0,C 180,E1 -23561.792,E2 -23561.792} C_VEL
LIN {X 0,Y 157.567,Z 385.858,A -85,B 0,C 180,E1 -23567.114,E2 -23567.114} C_VEL
LIN {X 0,Y 157.778,Z 385.832,A -85,B 0,C 180,E1 -23569.737,E2 -23569.737} C_VEL
LIN {X 0,Y 157.83,Z 385.825,A -85,B 0,C 180,E1 -23572.324,E2 -23572.324} C_VEL
LIN {X 0,Y 158.264,Z 385.759,A -85,B 0,C 180,E1 -23580.001,E2 -23580.001} C_VEL
LIN {X 0,Y 157.828,Z 385.808,A -85,B 0,C 180,E1 -23587.678,E2 -23587.678} C_VEL
LIN {X 0,Y 157.711,Z 385.839,A -85,B 0,C 180,E1 -23591.361,E2 -23591.361} C_VEL
LIN {X 0,Y 157.468,Z 385.853,A -85,B 0,C 180,E1 -23595.533,E2 -23595.533} C_VEL
LIN {X 0,Y 157.376,Z 385.877,A -85,B 0,C 180,E1 -23600.933,E2 -23600.933} C_VEL
LIN {X 0,Y 157.321,Z 385.888,A -85,B 0,C 180,E1 -23606.685,E2 -23606.685} C_VEL
LIN {X 0,Y 157.284,Z 385.891,A -85,B 0,C 180,E1 -23612.426,E2 -23612.426} C_VEL
LIN {X 0,Y 157.289,Z 385.891,A -85,B 0,C 180,E1 -23616.456,E2 -23616.456} C_VEL
LIN {X 0,Y 157.219,Z 385.897,A -85,B 0,C 180,E1 -23622.109,E2 -23622.109} C_VEL
LIN {X 0,Y 157.216,Z 385.897,A -85,B 0,C 180,E1 -23627.889,E2 -23627.889} C_VEL
LIN {X 0,Y 157.273,Z 385.893,A -85,B 0,C 180,E1 -23633.55,E2 -23633.55} C_VEL
LIN {X 0,Y 157.316,Z 385.887,A -85,B 0,C 180,E1 -23636.582,E2 -23636.582} C_VEL
LIN {X 0,Y 158.217,Z 388.541,A -85,B 0,C 180,E1 -23637.211,E2 -23637.211} C_VEL
LIN {X 0,Y 159.641,Z 390.867,A -85,B 0,C 180,E1 -23637.938,E2 -23637.938} C_VEL
LIN {X 0,Y 163.758,Z 399.268,A -85,B 0,C 180,E1 -23640.417,E2 -23640.417} C_VEL
LIN {X 0,Y 167.102,Z 407.271,A -85,B 0,C 180,E1 -23642.789,E2 -23642.789} C_VEL
LIN {X 0,Y 170.029,Z 416.631,A -85,B 0,C 180,E1 -23645.583,E2 -23645.583} C_VEL
LIN {X 0,Y 171.915,Z 424.343,A -85,B 0,C 180,E1 -23648.027,E2 -23648.027} C_VEL
LIN {X 0,Y 169.432,Z 434.108,A -85,B 0,C 180,E1 -23650.618,E2 -23650.618} C_VEL
LIN {X 0,Y 166.817,Z 442.821,A -85,B 0,C 180,E1 -23653.477,E2 -23653.477} C_VEL
LIN {X 0,Y 163.985,Z 451.353,A -85,B 0,C 180,E1 -23656.995,E2 -23656.995} C_VEL
LIN {X 0,Y 161.653,Z 458.167,A -85,B 0,C 180,E1 -23660.615,E2 -23660.615} C_VEL
LIN {X 0,Y 159.578,Z 464.434,A -85,B 0,C 180,E1 -23664.945,E2 -23664.945} C_VEL
LIN {X 0,Y 158.282,Z 468.568,A -85,B 0,C 180,E1 -23668.726,E2 -23668.726} C_VEL
LIN {X 0,Y 157.432,Z 471.676,A -85,B 0,C 180,E1 -23672.557,E2 -23672.557} C_VEL
LIN {X 0,Y 157.324,Z 473.214,A -85,B 0,C 180,E1 -23675.124,E2 -23675.124} C_VEL
LIN {X 0,Y 157.369,Z 474.321,A -85,B 0,C 180,E1 -23677.698,E2 -23677.698} C_VEL
LIN {X 0,Y 157.948,Z 475.397,A -85,B 0,C 180,E1 -23682.853,E2 -23682.853} C_VEL
LIN {X 0,Y 158.589,Z 475.367,A -85,B 0,C 180,E1 -23685.418,E2 -23685.418} C_VEL
LIN {X 0,Y 159.46,Z 474.908,A -85,B 0,C 180,E1 -23687.968,E2 -23687.968} C_VEL
LIN {X 0,Y 161.963,Z 472.801,A -85,B 0,C 180,E1 -23692.986,E2 -23692.986} C_VEL
LIN {X 0,Y 163.731,Z 470.954,A -85,B 0,C 180,E1 -23695.655,E2 -23695.655} C_VEL
LIN {X 0,Y 167.49,Z 466.375,A -85,B 0,C 180,E1 -23700.232,E2 -23700.232} C_VEL
LIN {X 0,Y 171.02,Z 461.495,A -85,B 0,C 180,E1 -23703.693,E2 -23703.693} C_VEL
LIN {X 0,Y 175.121,Z 455.291,A -85,B 0,C 180,E1 -23707.01,E2 -23707.01} C_VEL
LIN {X 0,Y 179.644,Z 447.448,A -85,B 0,C 180,E1 -23710.202,E2 -23710.202} C_VEL
LIN {X 0,Y 181.758,Z 443.412,A -85,B 0,C 180,E1 -23711.558,E2 -23711.558} C_VEL
LIN {X 0,Y 182.067,Z 442.409,A -85,B 0,C 180,E1 -23711.938,E2 -23711.938} C_VEL
LIN {X 0,Y 181.231,Z 435.417,A -85,B 0,C 180,E1 -23715.255,E2 -23715.255} C_VEL
LIN {X 0,Y 179.505,Z 427.767,A -85,B 0,C 180,E1 -23718.81,E2 -23718.81} C_VEL
LIN {X 0,Y 176.995,Z 419.68,A -85,B 0,C 180,E1 -23722.572,E2 -23722.572} C_VEL
LIN {X 0,Y 173.882,Z 412.419,A -85,B 0,C 180,E1 -23726.203,E2 -23726.203} C_VEL
LIN {X 0,Y 170.237,Z 405.278,A -85,B 0,C 180,E1 -23730.103,E2 -23730.103} C_VEL
LIN {X 0,Y 167.855,Z 401.149,A -85,B 0,C 180,E1 -23732.576,E2 -23732.576} C_VEL
LIN {X 0,Y 166.611,Z 399.702,A -85,B 0,C 180,E1 -23733.709,E2 -23733.709} C_VEL
LIN {X 0,Y 165.59,Z 397.712,A -85,B 0,C 180,E1 -23734.885,E2 -23734.885} C_VEL
LIN {X 0,Y 162.318,Z 393.412,A -85,B 0,C 180,E1 -23738.322,E2 -23738.322} C_VEL
LIN {X 0,Y 161.641,Z 391.508,A -85,B 0,C 180,E1 -23739.312,E2 -23739.312} C_VEL
LIN {X 0,Y 159.119,Z 389.617,A -85,B 0,C 180,E1 -23741.99,E2 -23741.99} C_VEL
LIN {X 0,Y 157.805,Z 387.323,A -85,B 0,C 180,E1 -23743.838,E2 -23743.838} C_VEL
LIN {X 0,Y 157.47,Z 385.868,A -85,B 0,C 180,E1 -23744.633,E2 -23744.633} C_VEL
LIN {X 0,Y 157.769,Z 385.827,A -85,B 0,C 180,E1 -23749.735,E2 -23749.735} C_VEL
LIN {X 0,Y 157.821,Z 385.817,A -85,B 0,C 180,E1 -23752.322,E2 -23752.322} C_VEL
LIN {X 0,Y 157.999,Z 385.804,A -85,B 0,C 180,E1 -23757.45,E2 -23757.45} C_VEL
LIN {X 0,Y 158.257,Z 385.753,A -85,B 0,C 180,E1 -23759.999,E2 -23759.999} C_VEL
LIN {X 0,Y 157.8,Z 385.929,A -85,B 0,C 180,E1 -23767.035,E2 -23767.035} C_VEL
LIN {X 0,Y 158.085,Z 387.112,A -85,B 0,C 180,E1 -23770.243,E2 -23770.243} C_VEL
LIN {X 0,Y 158.285,Z 389.54,A -85,B 0,C 180,E1 -23775.45,E2 -23775.45} C_VEL
LIN {X 0,Y 158.806,Z 392.312,A -85,B 0,C 180,E1 -23780.734,E2 -23780.734} C_VEL
LIN {X 0,Y 159.2,Z 394.73,A -85,B 0,C 180,E1 -23784.448,E2 -23784.448} C_VEL
LIN {X 0,Y 160.947,Z 398.785,A -85,B 0,C 180,E1 -23786.536,E2 -23786.536} C_VEL
LIN {X 0,Y 164.239,Z 403.224,A -85,B 0,C 180,E1 -23789.654,E2 -23789.654} C_VEL
LIN {X 0,Y 166.133,Z 407.511,A -85,B 0,C 180,E1 -23791.567,E2 -23791.567} C_VEL
LIN {X 0,Y 168.131,Z 410.547,A -85,B 0,C 180,E1 -23793.237,E2 -23793.237} C_VEL
LIN {X 0,Y 170.074,Z 415.083,A -85,B 0,C 180,E1 -23795.074,E2 -23795.074} C_VEL
LIN {X 0,Y 171.323,Z 417.554,A -85,B 0,C 180,E1 -23796.13,E2 -23796.13} C_VEL
LIN {X 0,Y 174.136,Z 424.522,A -85,B 0,C 180,E1 -23798.724,E2 -23798.724} C_VEL
LIN {X 0,Y 176.56,Z 431.151,A -85,B 0,C 180,E1 -23801.053,E2 -23801.053} C_VEL
LIN {X 0,Y 178.219,Z 437,A -85,B 0,C 180,E1 -23802.933,E2 -23802.933} C_VEL
LIN {X 0,Y 178.13,Z 448.309,A -85,B 0,C 180,E1 -23805.674,E2 -23805.674} C_VEL
LIN {X 0,Y 177.048,Z 460.077,A -85,B 0,C 180,E1 -23808.761,E2 -23808.761} C_VEL
LIN {X 0,Y 175.338,Z 469.758,A -85,B 0,C 180,E1 -23811.592,E2 -23811.592} C_VEL
LIN {X 0,Y 172.861,Z 479.5,A -85,B 0,C 180,E1 -23814.877,E2 -23814.877} C_VEL
LIN {X 0,Y 170.436,Z 486.389,A -85,B 0,C 180,E1 -23817.586,E2 -23817.586} C_VEL
LIN {X 0,Y 167.877,Z 491.514,A -85,B 0,C 180,E1 -23819.845,E2 -23819.845} C_VEL
LIN {X 0,Y 163.965,Z 497.896,A -85,B 0,C 180,E1 -23823.254,E2 -23823.254} C_VEL
LIN {X 0,Y 160.798,Z 503.041,A -85,B 0,C 180,E1 -23826.838,E2 -23826.838} C_VEL
LIN {X 0,Y 158.435,Z 507.098,A -85,B 0,C 180,E1 -23830.57,E2 -23830.57} C_VEL
LIN {X 0,Y 156.732,Z 510.151,A -85,B 0,C 180,E1 -23834.395,E2 -23834.395} C_VEL
LIN {X 0,Y 155.782,Z 512.785,A -85,B 0,C 180,E1 -23839.606,E2 -23839.606} C_VEL
LIN {X 0,Y 155.854,Z 513.634,A -85,B 0,C 180,E1 -23842.772,E2 -23842.772} C_VEL
LIN {X 0,Y 156.557,Z 513.782,A -85,B 0,C 180,E1 -23847.429,E2 -23847.429} C_VEL
